(* CFC diagram, written out as Structured Text *)
GVL.s3363[s3363_Mapping.ACV_203].PLC_CMD := RAMP_REAL_1.OUT;
_OR123_OUT := (PVL.Z202_Config.Status.eStatus=eZ202_Status.Recovery_Active_P202) OR (PVL.Z202_Config.Status.eStatus=eZ202_Status.Recovery_Active_P203) OR (PVL.Z202_Config.Status.eStatus=eZ202_Status.Fixed_Rate_Recovery_Active_P202) OR (PVL.Z202_Config.Status.eStatus=eZ202_Status.Fixed_Rate_Recovery_Active_P203) OR (PVL.Z202_Config.Status.eStatus=eZ202_Status.Continuous_Level_And_Recovery_Speed) OR (PVL.Z202_Config.Status.eStatus=eZ202_Status.Continuous_Flow_And_Recovery_Speed) OR (PVL.Z202_Config.Status.eStatus=eZ202_Status.Continuous_Level_And_Recovery_Flow) OR (PVL.Z202_Config.Status.eStatus=eZ202_Status.Continuous_Flow_And_Recovery_Flow);
GVL.s3363[s3363_mapping.ACV_225].PLC_CMD := SEL(PVl.Z202_Config.Valve_Pattern[SubIndex].Matrix.1 AND _OR123_OUT, 0.0, 100);
GVL.s3363[s3363_mapping.ACV_226].PLC_CMD := SEL(_AND161_OUT OR False OR False OR _AND185_OUT, 0.0, 100);
_OR66_OUT := (PVL.Z202_Config.Status.eStatus=eZ202_Status.Opening_ACV203) OR (PVL.Z202_Config.Status.eStatus=eZ202_Status.TK201_Level_Return_Via_P203) OR (PVL.Z202_Config.Status.eStatus=eZ202_Status.Fixed_Rate_Return_Via_P203) OR (PVL.Z202_Config.Status.eStatus=eZ202_Status.Fixed_Rate_Recovery_Active_P203) OR (PVL.Z202_Config.Status.eStatus=eZ202_Status.Recovery_Active_P203) OR (PVL.Z202_Config.Status.eStatus=eZ202_Status.Fixed_Rate_Recovery_Active_P203) OR (PVL.Z202_Config.Status.eStatus=eZ202_Status.Continuous_Level_And_Recovery_Speed) OR (PVL.Z202_Config.Status.eStatus=eZ202_Status.Continuous_Flow_And_Recovery_Speed) OR (PVL.Z202_Config.Status.eStatus=eZ202_Status.Continuous_Level_And_Recovery_Flow) OR (PVL.Z202_Config.Status.eStatus=eZ202_Status.Continuous_Flow_And_Recovery_Flow);
GVL.s3363[s3363_Mapping.ACV_206].PLC_CMD := RAMP_REAL_0.OUT;
RAMP_REAL_0(IN := SEL(_OR241_OUT, 0.0, 100), ASCEND := 50, DESCEND := 5, TIMEBASE := T#1s, RESET := False);
_AND185_OUT := _OR187_OUT AND _OR207_OUT;
_OR187_OUT := (PVL.Z202_Config.Task.eTask=eZ202_Task.TK201_Level_Return_P203) OR (PVL.Z202_Config.Task.eTask=eZ202_Task.Rate_Return_P203) OR (PVL.Z202_Config.Task.eTask=eZ202_Task.Filter_Flow_P203) OR (PVL.Z202_Config.Task.eTask=eZ202_Task.Filter_Level_P203) OR (PVL.Z202_Config.Task.eTask=eZ202_task.Filter_Level_P202_Recovery_Speed_P203) OR (PVL.Z202_Config.Task.eTask=eZ202_task.Filter_Level_P202_Recovery_Flow_P203) OR (PVL.Z202_Config.Task.eTask=eZ202_task.Filter_Flow_P202_Recovery_Speed_P203) OR (PVL.Z202_Config.Task.eTask=eZ202_task.Filter_Flow_P202_Recovery_Flow_P203) OR (PVL.Z202_Config.Task.eTask=eZ202_task.Drain_P203);
_OR48_OUT := (PVL.Z202_Config.Task.eTask=eZ202_Task.TK201_Level_Return_P203) OR (PVL.Z202_Config.Task.eTask=eZ202_Task.Rate_Return_P203) OR (PVL.Z202_Config.Task.eTask=eZ202_Task.Recovery_Rate_P203) OR (PVL.Z202_Config.Task.eTask=eZ202_Task.Recovery_Speed_P203) OR (PVL.Z202_Config.Task.eTask=eZ202_task.Filter_Level_P202_Recovery_Speed_P203) OR (PVL.Z202_Config.Task.eTask=eZ202_task.Filter_Level_P202_Recovery_Flow_P203) OR (PVL.Z202_Config.Task.eTask=eZ202_task.Filter_Flow_P202_Recovery_Speed_P203) OR (PVL.Z202_Config.Task.eTask=eZ202_task.Filter_Flow_P202_Recovery_Flow_P203);
_OR14_OUT := (PVL.Z202_Config.Task.eTask=eZ202_Task.TK201_Level_Return_P202) OR (PVL.Z202_Config.Task.eTask=eZ202_Task.Rate_Return_P202) OR (PVL.Z202_Config.Task.eTask=eZ202_Task.Recovery_Rate_P202) OR (PVL.Z202_Config.Task.eTask=eZ202_Task.Recovery_Speed_P202);
_OR24_OUT := (PVL.Z202_Config.Status.eStatus=eZ202_Status.Opening_ACV203) OR (PVL.Z202_Config.Status.eStatus=eZ202_Status.TK201_Level_Return_Via_P202) OR (PVL.Z202_Config.Status.eStatus=eZ202_Status.Fixed_Rate_Return_Via_P202) OR (PVL.Z202_Config.Status.eStatus=eZ202_Status.Recovery_Active_P202) OR (PVL.Z202_Config.Status.eStatus=eZ202_Status.Fixed_Rate_Recovery_Active_P202);
RAMP_REAL_1(IN := _SEL4_OUT, ASCEND := 50, DESCEND := 5, TIMEBASE := T#1s, RESET := False);
RS_ACV_203();
_SEL4_OUT := SEL((PVL.Z202_Config.Status.eStatus=eZ202_Status.EP101_Level_Return_Via_P203) OR (PVL.Z202_Config.Status.eStatus=eZ202_Status.EP101_Level_Return_Via_P202) OR _OR14_OUT AND _OR24_OUT OR False OR False OR False OR False OR False OR _OR48_OUT AND _OR66_OUT, 0.0, 100);
_OR241_OUT := (PVL.Z202_Config.Status.eStatus=eZ202_Status.EP101_Level_Return_Via_P202) OR False OR False OR False OR False OR _AND253_OUT;
_OR207_OUT := (PVL.Z202_Config.Status.eStatus=eZ202_Status.Opening_ACV206) OR (PVL.Z202_Config.Status.eStatus=eZ202_Status.Opening_ACV203) OR (PVL.Z202_Config.Status.eStatus=eZ202_Status.Opening_ACV226) OR (PVL.Z202_Config.Status.eStatus=eZ202_Status.Fixed_Rate_Return_Via_P203) OR (PVL.Z202_Config.Status.eStatus=eZ202_Status.TK201_Level_Return_Via_P203) OR (PVL.Z202_Config.Status.eStatus=eZ202_Status.Filters_TK201_Level_Control_P203) OR (PVL.Z202_Config.Status.eStatus=eZ202_Status.Filters_Fixed_Flow_Control_P203) OR (PVL.Z202_Config.Status.eStatus=eZ202_Status.Continuous_Level_And_Recovery_Speed) OR (PVL.Z202_Config.Status.eStatus=eZ202_Status.Continuous_Flow_And_Recovery_Speed) OR (PVL.Z202_Config.Status.eStatus=eZ202_Status.Continuous_Level_And_Recovery_Flow) OR (PVL.Z202_Config.Status.eStatus=eZ202_Status.Continuous_Flow_And_Recovery_Flow) OR (PVL.Z202_Config.Status.eStatus=eZ202_Status.Drain_Active_P203);
_AND253_OUT := _OR255_OUT AND _OR271_OUT;
_OR271_OUT := (PVL.Z202_Config.Status.eStatus=eZ202_Status.Opening_ACV206) OR (PVL.Z202_Config.Status.eStatus=eZ202_Status.Opening_ACV203) OR (PVL.Z202_Config.Status.eStatus=eZ202_Status.TK201_Level_Return_Via_P202) OR (PVL.Z202_Config.Status.eStatus=eZ202_Status.Fixed_Rate_Return_Via_P202) OR (PVL.Z202_Config.Status.eStatus=eZ202_Status.Recovery_Active_P202) OR (PVL.Z202_Config.Status.eStatus=eZ202_Status.Fixed_Rate_Recovery_Active_P202) OR (PVL.Z202_Config.Status.eStatus=eZ202_Status.Filters_Fixed_Flow_Control_P203) OR (PVL.Z202_Config.Status.eStatus=eZ202_Status.Filters_TK201_Level_Control_P203) OR (PVL.Z202_Config.Status.eStatus=eZ202_Status.Drain_Active_P203);
_OR255_OUT := (PVL.Z202_Config.Task.eTask=eZ202_Task.TK201_Level_Return_P202) OR (PVL.Z202_Config.Task.eTask=eZ202_Task.Rate_Return_P202) OR (PVL.Z202_Config.Task.eTask=eZ202_Task.Recovery_Rate_P202) OR (PVL.Z202_Config.Task.eTask=eZ202_Task.Recovery_Speed_P202) OR (PVL.Z202_Config.Task.eTask=eZ202_Task.Filter_Flow_P203) OR (PVL.Z202_Config.Task.eTask=eZ202_Task.Filter_Level_P203) OR (PVL.Z202_Config.Task.eTask=eZ202_Task.Drain_P203);
_AND161_OUT := ((PVL.Z202_Config.Task.eTask=eZ202_Task.TK201_Level_Return_P202) OR (PVL.Z202_Config.Task.eTask=eZ202_Task.Rate_Return_P202) OR (PVL.Z202_Config.Task.eTask=eZ202_Task.Filter_Level_P202) OR (PVL.Z202_Config.Task.eTask=eZ202_Task.Filter_Flow_P202) OR (PVL.Z202_Config.Task.eTask=eZ202_Task.Drain_P202)) AND _OR164_OUT;
_OR164_OUT := (PVL.Z202_Config.Status.eStatus=eZ202_Status.Opening_ACV206) OR (PVL.Z202_Config.Status.eStatus=eZ202_Status.Opening_ACV203) OR (PVL.Z202_Config.Status.eStatus=eZ202_Status.Opening_ACV226) OR (PVL.Z202_Config.Status.eStatus=eZ202_Status.TK201_Level_Return_Via_P202) OR (PVL.Z202_Config.Status.eStatus=eZ202_Status.Fixed_Rate_Return_Via_P202) OR (PVL.Z202_Config.Status.eStatus=eZ202_Status.Filters_TK201_Level_Control_P202) OR (PVL.Z202_Config.Status.eStatus=eZ202_Status.Filters_Fixed_Flow_Control_P202) OR (PVL.Z202_Config.Status.eStatus=eZ202_Status.Drain_Active_P202);
GVL.s3363[s3363_mapping.ACV_224].PLC_CMD := SEL(PVl.Z202_Config.Valve_Pattern[SubIndex].Matrix.0 AND ((PVL.Z202_Config.Status.eStatus=eZ202_Status.Recovery_Active_P202) OR (PVL.Z202_Config.Status.eStatus=eZ202_Status.Recovery_Active_P203) OR (PVL.Z202_Config.Status.eStatus=eZ202_Status.Fixed_Rate_Recovery_Active_P202) OR (PVL.Z202_Config.Status.eStatus=eZ202_Status.Fixed_Rate_Recovery_Active_P203) OR (PVL.Z202_Config.Status.eStatus=eZ202_Status.Continuous_Level_And_Recovery_Speed) OR (PVL.Z202_Config.Status.eStatus=eZ202_Status.Continuous_Flow_And_Recovery_Speed) OR (PVL.Z202_Config.Status.eStatus=eZ202_Status.Continuous_Level_And_Recovery_Flow) OR (PVL.Z202_Config.Status.eStatus=eZ202_Status.Continuous_Flow_And_Recovery_Flow)), 0.0, 100);
(* drawn but not wired to any output: PVL.PID[PID_Mapping.Z202_Flow].Actual>5, 50 *)
END_ACTION

ACTION Test_P202_Conflict:
                (*
CASE PVL.Z202_Config.P202_Task.eTask OF
	eZ202_Task.EP101_Level_Return_P202:
		CASE PVl.Z202_Config.P203_Task.eTask OF
			eZ202_Task.EP101_Level_Return_P203:PVL.Z202_Config.P203_Task.eTask:=eZ202_Task.Off;
			eZ202_Task.Filter_Flow_P203:
			eZ202_Task.Filter_Level_P203:
			eZ202_Task.Rate_Return_P203:PVL.Z202_Config.P203_Task.eTask:=eZ202_Task.Off;
			eZ202_Task.Recovery_Rate_P203:PVL.Z202_Config.P203_Task.eTask:=eZ202_Task.Off;
			eZ202_Task.Recovery_Speed_P203:PVL.Z202_Config.P203_Task.eTask:=eZ202_Task.Off;
			eZ202_Task.TK201_Level_Return_P203:PVL.Z202_Config.P203_Task.eTask:=eZ202_Task.Off;
		END_CASE
	eZ202_Task.Filter_Flow_P202:
		CASE PVl.Z202_Config.P203_Task.eTask OF
			eZ202_Task.EP101_Level_Return_P203:
			eZ202_Task.Filter_Flow_P203:PVL.Z202_Config.P203_Task.eTask:=eZ202_Task.Off;
			eZ202_Task.Filter_Level_P203:PVL.Z202_Config.P203_Task.eTask:=eZ202_Task.Off;
			eZ202_Task.Rate_Return_P203:
			eZ202_Task.Recovery_Rate_P203:
			eZ202_Task.Recovery_Speed_P203:
			eZ202_Task.TK201_Level_Return_P203:
		END_CASE
	eZ202_Task.Filter_Level_P202:
		CASE PVl.Z202_Config.P203_Task.eTask OF
			eZ202_Task.EP101_Level_Return_P203:
			eZ202_Task.Filter_Flow_P203:PVL.Z202_Config.P203_Task.eTask:=eZ202_Task.Off;
			eZ202_Task.Filter_Level_P203:PVL.Z202_Config.P203_Task.eTask:=eZ202_Task.Off;
			eZ202_Task.Rate_Return_P203:
			eZ202_Task.Recovery_Rate_P203:
			eZ202_Task.Recovery_Speed_P203:
			eZ202_Task.TK201_Level_Return_P203:
		END_CASE
	eZ202_Task.Rate_Return_P202:
		CASE PVl.Z202_Config.P203_Task.eTask OF
			eZ202_Task.EP101_Level_Return_P203:PVL.Z202_Config.P203_Task.eTask:=eZ202_Task.Off;
			eZ202_Task.Filter_Flow_P203:
			eZ202_Task.Filter_Level_P203:
			eZ202_Task.Rate_Return_P203:PVL.Z202_Config.P203_Task.eTask:=eZ202_Task.Off;
			eZ202_Task.Recovery_Rate_P203:PVL.Z202_Config.P203_Task.eTask:=eZ202_Task.Off;
			eZ202_Task.Recovery_Speed_P203:PVL.Z202_Config.P203_Task.eTask:=eZ202_Task.Off;
			eZ202_Task.TK201_Level_Return_P203:PVL.Z202_Config.P203_Task.eTask:=eZ202_Task.Off;
		END_CASE
	eZ202_Task.Recovery_Rate_P202:
		CASE PVl.Z202_Config.P203_Task.eTask OF
			eZ202_Task.EP101_Level_Return_P203:PVL.Z202_Config.P203_Task.eTask:=eZ202_Task.Off;
			eZ202_Task.Filter_Flow_P203:
			eZ202_Task.Filter_Level_P203:
			eZ202_Task.Rate_Return_P203:PVL.Z202_Config.P203_Task.eTask:=eZ202_Task.Off;
			eZ202_Task.Recovery_Rate_P203:PVL.Z202_Config.P203_Task.eTask:=eZ202_Task.Off;
			eZ202_Task.Recovery_Speed_P203:PVL.Z202_Config.P203_Task.eTask:=eZ202_Task.Off;
			eZ202_Task.TK201_Level_Return_P203:PVL.Z202_Config.P203_Task.eTask:=eZ202_Task.Off;
		END_CASE
	eZ202_Task.Recovery_Speed_P202:
		CASE PVl.Z202_Config.P203_Task.eTask OF
			eZ202_Task.EP101_Level_Return_P203:PVL.Z202_Config.P203_Task.eTask:=eZ202_Task.Off;
			eZ202_Task.Filter_Flow_P203:
			eZ202_Task.Filter_Level_P203:
			eZ202_Task.Rate_Return_P203:PVL.Z202_Config.P203_Task.eTask:=eZ202_Task.Off;
			eZ202_Task.Recovery_Rate_P203:PVL.Z202_Config.P203_Task.eTask:=eZ202_Task.Off;
			eZ202_Task.Recovery_Speed_P203:PVL.Z202_Config.P203_Task.eTask:=eZ202_Task.Off;
			eZ202_Task.TK201_Level_Return_P203:PVL.Z202_Config.P203_Task.eTask:=eZ202_Task.Off;
		END_CASE
	eZ202_Task.TK201_Level_Return_P202:
		CASE PVl.Z202_Config.P203_Task.eTask OF
			eZ202_Task.EP101_Level_Return_P203:PVL.Z202_Config.P203_Task.eTask:=eZ202_Task.Off;
			eZ202_Task.Filter_Flow_P203:
			eZ202_Task.Filter_Level_P203:
			eZ202_Task.Rate_Return_P203:PVL.Z202_Config.P203_Task.eTask:=eZ202_Task.Off;
			eZ202_Task.Recovery_Rate_P203:PVL.Z202_Config.P203_Task.eTask:=eZ202_Task.Off;
			eZ202_Task.Recovery_Speed_P203:PVL.Z202_Config.P203_Task.eTask:=eZ202_Task.Off;
			eZ202_Task.TK201_Level_Return_P203:PVL.Z202_Config.P203_Task.eTask:=eZ202_Task.Off;
		END_CASE
	
END_CASE
*)

              
END_ACTION

ACTION Rate_Return_P202:
                IF PVL.Z202_Config.Task.eTask<> Local_Task THEN
	Local_Task:=PVL.Z202_Config.Task.eTask;
	SubIndex:=0;
	Task_ton.IN:=FALSE;
	local_Status:=eZ202_Status.Opening_Valves;
	PVL.Filter_Config.Mode.eMode:=eFilter_Mode.Off;
	PVL.Z202_Config.ETA:=0;
	Level_Ton.PT:=T#10S;
END_IF;

PVL.PID[PID_Mapping.Z202_Flow].PLC_Target:=PVL.Z202_Config.TK201_Return_Rate.Target;




CASE PVL.Z202_Config.Status.eStatus OF
	eZ202_status.Opening_Valves:
		Local_Status:=eZ202_Status.Opening_ACV226;
	eZ202_status.Opening_ACV226:
		IF GVL.s3363[s3363_mapping.ACV_226].Valve_Actual>75 THEN	Local_Status:=eZ202_Status.Opening_ACV206; END_IF;
	eZ202_Status.Opening_ACV206:
		IF GVL.s3363[s3363_Mapping.ACV_206].Valve_Actual>75 THEN Local_Status:=eZ202_Status.Opening_ACV203;END_IF;
	eZ202_Status.Opening_ACV203:
		IF GVL.s3363[s3363_mapping.ACV_203].Valve_Actual>75 THEN local_Status:=eZ202_Status.Fixed_Rate_Return_Via_P202; END_IF;
		
	eZ202_Status.LT101_High_High_Alarm:		IF Level_ton.Q THEN Local_Status:=eZ202_Status.Waiting_For_Level_OK_LT101; END_IF;
	eZ202_Status.LT201_High_High_Alarm:		IF Level_ton.Q THEN Local_Status:=eZ202_Status.Waiting_For_Level_OK_LT201; END_IF;
	eZ202_Status.LT202_Low_Low_Alarm:		IF Level_ton.Q THEN Local_Status:=eZ202_Status.Waiting_For_Level_OK_LT202; END_IF;
	
	
	eZ202_Status.Waiting_For_Level_OK_LT101:	IF PVL.AIT[ait_Mapping.LT_101_P].Status.eStatus=Burkert.eSensor_Status.OK THEN local_Status:=eZ202_Status.Opening_Valves; END_IF;
	eZ202_Status.Waiting_For_Level_OK_LT201:	IF PVL.AIT[ait_Mapping.LT_201].Status.eStatus=Burkert.eSensor_Status.OK THEN local_Status:=eZ202_Status.Opening_Valves; END_IF;
	eZ202_Status.Waiting_For_Level_OK_LT202:	IF PVL.AIT[ait_Mapping.LT_202].Status.eStatus=Burkert.eSensor_Status.OK THEN local_Status:=eZ202_Status.Opening_Valves; END_IF;

END_CASE;





PVL.Z202_Config.Status.eStatus:= Test_Z201_Return_P202(Local_Status);

Status_hold();



	
		
              
END_ACTION

ACTION Recovery_Rate_P202:
                IF PVL.Z202_Config.Task.eTask<> Local_Task THEN
	Local_Task:=PVL.Z202_Config.Task.eTask;
	SubIndex:=0;
	Task_ton.IN:=FALSE;
	Valve_Ton.IN:=FALSE;
	local_Status:=eZ202_Status.Opening_Valves;
END_IF;



PVL.PID[PID_Mapping.Z202_Flow].PLC_Target:=PVL.Z202_Config.Recovery_Rate.Target;

	
	



Task_ton.PT:=TO_TIME(PVL.Z202_Config.Recovery_Duration_Min);	
Task_ton.IN:=PVL.Z202_Config.Status.eStatus=eZ202_Status.Fixed_Rate_Recovery_Active_P202;
	
//Valve_ton.PT:=TO_TIME(PVL.Z202_Config.Valve_Pattern[SubIndex].Duration);
//IF Valve_ton.Q THEN SubIndex:= ((SubIndex+1) MOD 5); END_IF;;
//Valve_Ton.IN:=NOT(Valve_Ton.Q);

CASE PVL.Z202_Config.Status.eStatus OF
	eZ202_status.Opening_Valves:
		Local_Status:=eZ202_Status.Opening_ACV206;
	eZ202_status.Opening_ACV226:
		IF GVL.s3363[s3363_mapping.ACV_226].Valve_Actual>75 THEN	Local_Status:=eZ202_Status.Opening_ACV206; END_IF;
	eZ202_Status.Opening_ACV206:
		IF GVL.s3363[s3363_Mapping.ACV_206].Valve_Actual>75 THEN Local_Status:=eZ202_Status.Opening_ACV203;END_IF;
	eZ202_Status.Opening_ACV203:
		IF GVL.s3363[s3363_mapping.ACV_203].Valve_Actual>75 THEN local_Status:=eZ202_Status.Fixed_Rate_Recovery_Active_P202; END_IF;
	eZ202_Status.Fixed_Rate_Recovery_Active_P202:
		IF Task_Ton.Q THEN	Local_Status:=eZ202_Status.Recovery_P202_Complete;	END_IF;
	eZ202_Status.LT101_High_High_Alarm:		IF Level_ton.Q THEN Local_Status:=eZ202_Status.Waiting_For_Level_OK_LT101; END_IF;
	eZ202_Status.LT201_High_High_Alarm:		IF Level_ton.Q THEN Local_Status:=eZ202_Status.Waiting_For_Level_OK_LT201; END_IF;
	eZ202_Status.LT202_Low_Low_Alarm:		IF Level_ton.Q THEN Local_Status:=eZ202_Status.Waiting_For_Level_OK_LT202; END_IF;
	eZ202_Status.Waiting_For_Level_OK_LT101:	IF PVL.AIT[ait_Mapping.LT_101_P].Status.eStatus=Burkert.eSensor_Status.OK THEN Local_Task:=eZ202_Task.Off; END_IF;
	eZ202_Status.Waiting_For_Level_OK_LT201:	IF PVL.AIT[ait_Mapping.LT_201].Status.eStatus=Burkert.eSensor_Status.OK THEN Local_Task:=eZ202_Task.Off; END_IF;
	eZ202_Status.Waiting_For_Level_OK_LT202:	IF PVL.AIT[ait_Mapping.LT_202].Status.eStatus=Burkert.eSensor_Status.OK THEN Local_Task:=eZ202_Task.Off; END_IF;
		
END_CASE;



PVL.Z202_Config.Status.eStatus:= Test_All(Local_Status);
Status_hold();
              
END_ACTION

ACTION Status_Hold:
                CASE PVL.Z202_Config.Status.eStatus OF
	eZ202_Status.EP101_High_High_Alarm:		local_Status:=PVL.Z202_Config.Status.eStatus;
	eZ202_Status.P202_Intake_Empty:			local_Status:=PVL.Z202_Config.Status.eStatus;
	eZ202_Status.P203_Intake_Empty:			local_Status:=PVL.Z202_Config.Status.eStatus;
	eZ202_Status.PT202_High_Pressure_Alarm:		local_Status:=PVL.Z202_Config.Status.eStatus;
	eZ202_Status.PT202_Low_Pressure_Alarm:		local_Status:=PVL.Z202_Config.Status.eStatus;
	eZ202_Status.PT203_high_Pressure_Alarm:		local_Status:=PVL.Z202_Config.Status.eStatus;
	eZ202_Status.PT203_Low_Pressure_Alarm:		local_Status:=PVL.Z202_Config.Status.eStatus;
	eZ202_Status.PT202_Not_Ready:				local_Status:=PVL.Z202_Config.Status.eStatus;
	eZ202_Status.PT203_Not_Ready:				local_Status:=PVL.Z202_Config.Status.eStatus;
	eZ202_Status.LT202_Not_Ready:				local_Status:=PVL.Z202_Config.Status.eStatus;
	eZ202_Status.LT202A_Not_Ready:				local_Status:=PVL.Z202_Config.Status.eStatus;
	
	eZ202_Status.FT202_High_High_Flow_Alarm:				local_Status:=PVL.Z202_Config.Status.eStatus;
	ez202_Status.FT202_Low_Low_Flow_Alarm:				local_Status:=PVL.Z202_Config.Status.eStatus;
	eZ202_Status.FT203_High_High_Flow_Alarm:				local_Status:=PVL.Z202_Config.Status.eStatus;
	eZ202_Status.FT203_Low_Low_Flow_Alarm:				local_Status:=PVL.Z202_Config.Status.eStatus;
	//eZ202_Status.PT202_High_Pressure_Alarm:				local_Status:=PVL.Z202_Config.Status.eStatus;
	//eZ202_Status.PT202_Low_Pressure_Alarm:				local_Status:=PVL.Z202_Config.Status.eStatus;
	//eZ202_Status.PT203_High_Pressure_Alarm:				local_Status:=PVL.Z202_Config.Status.eStatus;
	//eZ202_Status.PT203_Low_Pressure_Alarm:					local_Status:=PVL.Z202_Config.Status.eStatus;



END_CASE
              
END_ACTION

ACTION Filter_Flow_P202_Recovery_Speed_P203:
                IF PVL.Z202_Config.Task.eTask<> Local_Task THEN
	Local_Task:=PVL.Z202_Config.Task.eTask;
	local_status:=eZ202_Status.Opening_ACV226;
END_IF;


PVL.PID[PID_Mapping.Z202_TK201_Level].PLC_Target:=PVL.Z202_Config.Filter_Level.Target;
PVL.PID[PID_Mapping.Z202_Filter_Flow ].PLC_Target:=PVL.Z202_Config.Filter_Rate.Target;









CASE PVL.Z202_Config.Status.eStatus OF
	eZ202_Status.Opening_ACV226:
		IF GVL.s3363[s3363_mapping.ACV_226].Valve_Actual>75 THEN	Local_Status:=eZ202_Status.Opening_ACV203;	END_IF;
	eZ202_Status.Opening_ACV203:
		IF GVL.s3363[s3363_Mapping.ACV_203].Valve_Actual>75 THEN	local_Status:=eZ202_Status.Continuous_Flow_And_Recovery_Speed; END_IF;
	eZ202_Status.Continuous_Flow_And_Recovery_Speed:
		IF Task_Ton.Q THEN	PVL.Z202_Config.Task.eTask:=eZ202_Task.Filter_Flow_P202;	END_IF;
	eZ202_Status.LT101_High_High_Alarm:		IF Level_ton.Q THEN Local_Status:=eZ202_Status.Waiting_For_Level_OK_LT101; END_IF;
	eZ202_Status.LT201_High_High_Alarm:		IF Level_ton.Q THEN Local_Status:=eZ202_Status.Waiting_For_Level_OK_LT201; END_IF;
	eZ202_Status.LT202_Low_Low_Alarm:		IF Level_ton.Q THEN Local_Status:=eZ202_Status.Waiting_For_Level_OK_LT202; END_IF;
	eZ202_Status.Waiting_For_Level_OK_LT101:	IF PVL.AIT[ait_Mapping.LT_101_P].Status.eStatus=Burkert.eSensor_Status.OK THEN Local_Task:=eZ202_Task.Off; END_IF;
	eZ202_Status.Waiting_For_Level_OK_LT201:	IF PVL.AIT[ait_Mapping.LT_201].Status.eStatus=Burkert.eSensor_Status.OK THEN Local_Task:=eZ202_Task.Off; END_IF;
	eZ202_Status.Waiting_For_Level_OK_LT202:	IF PVL.AIT[ait_Mapping.LT_202].Status.eStatus=Burkert.eSensor_Status.OK THEN Local_Task:=eZ202_Task.Off; END_IF;

END_CASE




 

//PVL.Z202_Config.Status.eStatus:= Test_Filters(Local_Status);



Task_ton.PT:=TO_TIME(PVL.Z202_Config.Recovery_Duration_Min);	
Task_ton.IN:=PVL.Z202_Config.Status.eStatus=eZ202_Status.Continuous_Flow_And_Recovery_Speed;
	
//Valve_ton.PT:=TO_TIME(PVL.Z202_Config.Valve_Pattern[SubIndex].Duration);
//IF Valve_ton.Q THEN SubIndex:= ((SubIndex+1) MOD 5); END_IF;;
//Valve_Ton.IN:=NOT(Valve_Ton.Q);



PVL.Z202_Config.Status.eStatus:= Test_Combined(local_Status);

Status_hold();
              
END_ACTION

ACTION Filter_Flow_P202_Recovery_Flow_P203:
                IF PVL.Z202_Config.Task.eTask<> Local_Task THEN
	Local_Task:=PVL.Z202_Config.Task.eTask;
	local_status:=eZ202_Status.Opening_ACV226;
END_IF;


PVL.PID[PID_Mapping.Z202_Flow].PLC_Target:=PVL.Z202_Config.Recovery_Rate.Target;
PVL.PID[PID_Mapping.Z202_Filter_Flow ].PLC_Target:=PVL.Z202_Config.Filter_Rate.Target;









CASE PVL.Z202_Config.Status.eStatus OF
	eZ202_Status.Opening_ACV226:
		IF GVL.s3363[s3363_mapping.ACV_226].Valve_Actual>75 THEN	Local_Status:=eZ202_Status.Opening_ACV203;	END_IF;
	eZ202_Status.Opening_ACV203:
		IF GVL.s3363[s3363_Mapping.ACV_203].Valve_Actual>75 THEN	local_Status:=eZ202_Status.Continuous_Flow_And_Recovery_Speed; END_IF;
	eZ202_Status.Continuous_Flow_And_Recovery_Speed:
		IF Task_Ton.Q THEN	PVL.Z202_Config.Task.eTask:=eZ202_Task.Filter_Flow_P202;	END_IF;
		
	eZ202_Status.LT101_High_High_Alarm:		IF Level_ton.Q THEN Local_Status:=eZ202_Status.Waiting_For_Level_OK_LT101; END_IF;
	eZ202_Status.LT201_High_High_Alarm:		IF Level_ton.Q THEN Local_Status:=eZ202_Status.Waiting_For_Level_OK_LT201; END_IF;
	eZ202_Status.LT202_Low_Low_Alarm:		IF Level_ton.Q THEN Local_Status:=eZ202_Status.Waiting_For_Level_OK_LT202; END_IF;
	eZ202_Status.Waiting_For_Level_OK_LT101:	IF PVL.AIT[ait_Mapping.LT_101_P].Status.eStatus=Burkert.eSensor_Status.OK THEN Local_Task:=eZ202_Task.Off; END_IF;
	eZ202_Status.Waiting_For_Level_OK_LT201:	IF PVL.AIT[ait_Mapping.LT_201].Status.eStatus=Burkert.eSensor_Status.OK THEN Local_Task:=eZ202_Task.Off; END_IF;
	eZ202_Status.Waiting_For_Level_OK_LT202:	IF PVL.AIT[ait_Mapping.LT_202].Status.eStatus=Burkert.eSensor_Status.OK THEN Local_Task:=eZ202_Task.Off; END_IF;

END_CASE




 





Task_ton.PT:=TO_TIME(PVL.Z202_Config.Recovery_Duration_Min);	
Task_ton.IN:=PVL.Z202_Config.Status.eStatus=eZ202_Status.Recovery_Active_P203;
	





PVL.Z202_Config.Status.eStatus:= Test_Combined(local_Status);



Status_hold();
              
END_ACTION

ACTION Alarms:
                PVL.Z202_Config.READY:=(Local_Status=PVl.Z202_Config.Status.eStatus);

CASE PVL.Z202_Config.Task.eTask OF
	eZ202_task.Off:
		PVL.AIT[AIT_Mapping.LT_202A].Alarm_Config.Silence:=FALSE;
		PVL.AIT[AIT_MApping.LT_202].Alarm_Config.Silence:=FALSE;
		PVL.s8312[s8312_mapping.PT_202].Alarm_Config.Silence:=TRUE;
		PVL.s8312[s8312_mapping.PT_203].Alarm_Config.Silence:=TRUE;
		PVL.s8050[s8050_mapping.FT_203A].CND.Alarm_Config.Silence:=TRUE;
		PVL.s8050[s8050_mapping.FT_203A].Temp.Alarm_Config.Silence:=TRUE;
		PVL.s8098[s8098_Mapping.FT_202].PDO.Concentration_1.Alarm_Config.Silence:=TRUE;
		PVL.s8098[s8098_Mapping.FT_202].PDO.Concentration_2.Alarm_Config.Silence:=TRUE;
		PVL.s8098[s8098_Mapping.FT_202].PDO.Totaliser_1.Alarm_Config.Silence:=TRUE;
		PVL.s8098[s8098_Mapping.FT_202].PDO.Totaliser_2.Alarm_Config.Silence:=TRUE;
		PVL.s8098[s8098_Mapping.FT_202].PDO.Temp.Alarm_Config.Silence:=TRUE;
		PVL.s8098[s8098_Mapping.FT_202].PDO.VolumeFlow.Alarm_Config.Silence:=TRUE;
		PVL.s8098[s8098_Mapping.FT_203].PDO.Concentration_1.Alarm_Config.Silence:=TRUE;
		PVL.s8098[s8098_Mapping.FT_203].PDO.Concentration_2.Alarm_Config.Silence:=TRUE;
		PVL.s8098[s8098_Mapping.FT_203].PDO.Totaliser_1.Alarm_Config.Silence:=TRUE;
		PVL.s8098[s8098_Mapping.FT_203].PDO.Totaliser_2.Alarm_Config.Silence:=TRUE;
		PVL.s8098[s8098_Mapping.FT_203].PDO.Temp.Alarm_Config.Silence:=TRUE;
		PVL.s8098[s8098_Mapping.FT_203].PDO.VolumeFlow.Alarm_Config.Silence:=TRUE;
	eZ202_Task.Drain_P202:
		PVL.AIT[AIT_Mapping.LT_202A].Alarm_Config.Silence:=FALSE;
		PVL.AIT[AIT_MApping.LT_202].Alarm_Config.Silence:=FALSE;
		PVL.s8312[s8312_mapping.PT_202].Alarm_Config.Silence:=(network.VFD[VFD_Mapping.VFD_202].Output_Pct<Min_Pump_Speed);
		PVL.s8312[s8312_mapping.PT_203].Alarm_Config.Silence:=TRUE;			
		PVL.s8050[s8050_mapping.FT_203A].CND.Alarm_Config.Silence:=TRUE;
		PVL.s8050[s8050_mapping.FT_203A].Temp.Alarm_Config.Silence:=TRUE;
		PVL.s8098[s8098_Mapping.FT_202].PDO.Concentration_1.Alarm_Config.Silence:=TRUE;
		PVL.s8098[s8098_Mapping.FT_202].PDO.Concentration_2.Alarm_Config.Silence:=TRUE;
		PVL.s8098[s8098_Mapping.FT_202].PDO.Totaliser_1.Alarm_Config.Silence:=TRUE;
		PVL.s8098[s8098_Mapping.FT_202].PDO.Totaliser_2.Alarm_Config.Silence:=TRUE;
		PVL.s8098[s8098_Mapping.FT_202].PDO.Temp.Alarm_Config.Silence:=TRUE;
		PVL.s8098[s8098_Mapping.FT_202].PDO.VolumeFlow.Alarm_Config.Silence:=(network.VFD[VFD_Mapping.VFD_202].Output_Pct<Min_Pump_Speed);
		PVL.s8098[s8098_Mapping.FT_203].PDO.Concentration_1.Alarm_Config.Silence:=TRUE;
		PVL.s8098[s8098_Mapping.FT_203].PDO.Concentration_2.Alarm_Config.Silence:=TRUE;
		PVL.s8098[s8098_Mapping.FT_203].PDO.Totaliser_1.Alarm_Config.Silence:=TRUE;
		PVL.s8098[s8098_Mapping.FT_203].PDO.Totaliser_2.Alarm_Config.Silence:=TRUE;
		PVL.s8098[s8098_Mapping.FT_203].PDO.Temp.Alarm_Config.Silence:=TRUE;
		PVL.s8098[s8098_Mapping.FT_203].PDO.VolumeFlow.Alarm_Config.Silence:=TRUE;
	eZ202_Task.Drain_P203:
		PVL.AIT[AIT_Mapping.LT_202A].Alarm_Config.Silence:=FALSE;
		PVL.AIT[AIT_MApping.LT_202].Alarm_Config.Silence:=FALSE;
		PVL.s8312[s8312_mapping.PT_202].Alarm_Config.Silence:=(network.VFD[VFD_Mapping.VFD_203].Output_Pct<Min_Pump_Speed);
		PVL.s8312[s8312_mapping.PT_203].Alarm_Config.Silence:=TRUE;			
		PVL.s8050[s8050_mapping.FT_203A].CND.Alarm_Config.Silence:=TRUE;
		PVL.s8050[s8050_mapping.FT_203A].Temp.Alarm_Config.Silence:=TRUE;
		PVL.s8098[s8098_Mapping.FT_202].PDO.Concentration_1.Alarm_Config.Silence:=TRUE;
		PVL.s8098[s8098_Mapping.FT_202].PDO.Concentration_2.Alarm_Config.Silence:=TRUE;
		PVL.s8098[s8098_Mapping.FT_202].PDO.Totaliser_1.Alarm_Config.Silence:=TRUE;
		PVL.s8098[s8098_Mapping.FT_202].PDO.Totaliser_2.Alarm_Config.Silence:=TRUE;
		PVL.s8098[s8098_Mapping.FT_202].PDO.Temp.Alarm_Config.Silence:=TRUE;
		PVL.s8098[s8098_Mapping.FT_202].PDO.VolumeFlow.Alarm_Config.Silence:=(network.VFD[VFD_Mapping.VFD_203].Output_Pct<Min_Pump_Speed);
		PVL.s8098[s8098_Mapping.FT_203].PDO.Concentration_1.Alarm_Config.Silence:=TRUE;
		PVL.s8098[s8098_Mapping.FT_203].PDO.Concentration_2.Alarm_Config.Silence:=TRUE;
		PVL.s8098[s8098_Mapping.FT_203].PDO.Totaliser_1.Alarm_Config.Silence:=TRUE;
		PVL.s8098[s8098_Mapping.FT_203].PDO.Totaliser_2.Alarm_Config.Silence:=TRUE;
		PVL.s8098[s8098_Mapping.FT_203].PDO.Temp.Alarm_Config.Silence:=TRUE;
		PVL.s8098[s8098_Mapping.FT_203].PDO.VolumeFlow.Alarm_Config.Silence:=TRUE;
	eZ202_Task.EP101_Level_Return_P202:
	eZ202_Task.EP101_Level_Return_P203:
	eZ202_Task.Filter_Flow_P202:
		PVL.AIT[AIT_Mapping.LT_202A].Alarm_Config.Silence:=FALSE;
		PVL.AIT[AIT_MApping.LT_202].Alarm_Config.Silence:=FALSE;
		PVL.s8312[s8312_mapping.PT_202].Alarm_Config.Silence:=(network.VFD[VFD_Mapping.VFD_202].Output_Pct<Min_Pump_Speed);
		PVL.s8312[s8312_mapping.PT_203].Alarm_Config.Silence:=TRUE;
			
		PVL.s8050[s8050_mapping.FT_203A].CND.Alarm_Config.Silence:=TRUE;
		PVL.s8050[s8050_mapping.FT_203A].Temp.Alarm_Config.Silence:=TRUE;
		
		PVL.s8098[s8098_Mapping.FT_202].PDO.Concentration_1.Alarm_Config.Silence:=TRUE;
		PVL.s8098[s8098_Mapping.FT_202].PDO.Concentration_2.Alarm_Config.Silence:=TRUE;
		PVL.s8098[s8098_Mapping.FT_202].PDO.Totaliser_1.Alarm_Config.Silence:=TRUE;
		PVL.s8098[s8098_Mapping.FT_202].PDO.Totaliser_2.Alarm_Config.Silence:=TRUE;
		PVL.s8098[s8098_Mapping.FT_202].PDO.Temp.Alarm_Config.Silence:=TRUE;
		PVL.s8098[s8098_Mapping.FT_202].PDO.VolumeFlow.Alarm_Config.Silence:=(network.VFD[VFD_Mapping.VFD_202].Output_Pct<Min_Pump_Speed);
		
		PVL.s8098[s8098_Mapping.FT_203].PDO.Concentration_1.Alarm_Config.Silence:=TRUE;
		PVL.s8098[s8098_Mapping.FT_203].PDO.Concentration_2.Alarm_Config.Silence:=TRUE;
		PVL.s8098[s8098_Mapping.FT_203].PDO.Totaliser_1.Alarm_Config.Silence:=TRUE;
		PVL.s8098[s8098_Mapping.FT_203].PDO.Totaliser_2.Alarm_Config.Silence:=TRUE;
		PVL.s8098[s8098_Mapping.FT_203].PDO.Temp.Alarm_Config.Silence:=TRUE;
		PVL.s8098[s8098_Mapping.FT_203].PDO.VolumeFlow.Alarm_Config.Silence:=TRUE;
	eZ202_Task.Filter_Flow_P203:
		PVL.AIT[AIT_Mapping.LT_202A].Alarm_Config.Silence:=FALSE;
		PVL.AIT[AIT_MApping.LT_202].Alarm_Config.Silence:=FALSE;
		PVL.s8312[s8312_mapping.PT_202].Alarm_Config.Silence:=(network.VFD[VFD_Mapping.VFD_203].Output_Pct<Min_Pump_Speed);
		PVL.s8312[s8312_mapping.PT_203].Alarm_Config.Silence:=TRUE;
			
		PVL.s8050[s8050_mapping.FT_203A].CND.Alarm_Config.Silence:=TRUE;
		PVL.s8050[s8050_mapping.FT_203A].Temp.Alarm_Config.Silence:=TRUE;
		
		PVL.s8098[s8098_Mapping.FT_202].PDO.Concentration_1.Alarm_Config.Silence:=TRUE;
		PVL.s8098[s8098_Mapping.FT_202].PDO.Concentration_2.Alarm_Config.Silence:=TRUE;
		PVL.s8098[s8098_Mapping.FT_202].PDO.Totaliser_1.Alarm_Config.Silence:=TRUE;
		PVL.s8098[s8098_Mapping.FT_202].PDO.Totaliser_2.Alarm_Config.Silence:=TRUE;
		PVL.s8098[s8098_Mapping.FT_202].PDO.Temp.Alarm_Config.Silence:=TRUE;
		PVL.s8098[s8098_Mapping.FT_202].PDO.VolumeFlow.Alarm_Config.Silence:=(network.VFD[VFD_Mapping.VFD_203].Output_Pct<Min_Pump_Speed);
		
		PVL.s8098[s8098_Mapping.FT_203].PDO.Concentration_1.Alarm_Config.Silence:=TRUE;
		PVL.s8098[s8098_Mapping.FT_203].PDO.Concentration_2.Alarm_Config.Silence:=TRUE;
		PVL.s8098[s8098_Mapping.FT_203].PDO.Totaliser_1.Alarm_Config.Silence:=TRUE;
		PVL.s8098[s8098_Mapping.FT_203].PDO.Totaliser_2.Alarm_Config.Silence:=TRUE;
		PVL.s8098[s8098_Mapping.FT_203].PDO.Temp.Alarm_Config.Silence:=TRUE;
		PVL.s8098[s8098_Mapping.FT_203].PDO.VolumeFlow.Alarm_Config.Silence:=TRUE;
		
	eZ202_Task.Filter_Level_P202:
		PVL.AIT[AIT_Mapping.LT_202A].Alarm_Config.Silence:=FALSE;
		PVL.AIT[AIT_MApping.LT_202].Alarm_Config.Silence:=FALSE;
		PVL.s8312[s8312_mapping.PT_202].Alarm_Config.Silence:=(network.VFD[VFD_Mapping.VFD_202].Output_Pct<Min_Pump_Speed);
		PVL.s8312[s8312_mapping.PT_203].Alarm_Config.Silence:=TRUE;
		PVL.s8050[s8050_mapping.FT_203A].CND.Alarm_Config.Silence:=TRUE;
		PVL.s8050[s8050_mapping.FT_203A].Temp.Alarm_Config.Silence:=TRUE;
		PVL.s8098[s8098_Mapping.FT_202].PDO.Concentration_1.Alarm_Config.Silence:=TRUE;
		PVL.s8098[s8098_Mapping.FT_202].PDO.Concentration_2.Alarm_Config.Silence:=TRUE;
		PVL.s8098[s8098_Mapping.FT_202].PDO.Totaliser_1.Alarm_Config.Silence:=TRUE;
		PVL.s8098[s8098_Mapping.FT_202].PDO.Totaliser_2.Alarm_Config.Silence:=TRUE;
		PVL.s8098[s8098_Mapping.FT_202].PDO.Temp.Alarm_Config.Silence:=TRUE;
		PVL.s8098[s8098_Mapping.FT_202].PDO.VolumeFlow.Alarm_Config.Silence:=TRUE;//(network.VFD[VFD_Mapping.VFD_202].Output_Pct<Min_Pump_Speed);
		PVL.s8098[s8098_Mapping.FT_203].PDO.Concentration_1.Alarm_Config.Silence:=TRUE;
		PVL.s8098[s8098_Mapping.FT_203].PDO.Concentration_2.Alarm_Config.Silence:=TRUE;
		PVL.s8098[s8098_Mapping.FT_203].PDO.Totaliser_1.Alarm_Config.Silence:=TRUE;
		PVL.s8098[s8098_Mapping.FT_203].PDO.Totaliser_2.Alarm_Config.Silence:=TRUE;
		PVL.s8098[s8098_Mapping.FT_203].PDO.Temp.Alarm_Config.Silence:=TRUE;
		PVL.s8098[s8098_Mapping.FT_203].PDO.VolumeFlow.Alarm_Config.Silence:=TRUE;
	eZ202_Task.Filter_Level_P203:
		PVL.AIT[AIT_Mapping.LT_202A].Alarm_Config.Silence:=FALSE;
		PVL.AIT[AIT_MApping.LT_202].Alarm_Config.Silence:=FALSE;
		PVL.s8312[s8312_mapping.PT_202].Alarm_Config.Silence:=(network.VFD[VFD_Mapping.VFD_203].Output_Pct<Min_Pump_Speed);
		PVL.s8312[s8312_mapping.PT_203].Alarm_Config.Silence:=TRUE;
		PVL.s8050[s8050_mapping.FT_203A].CND.Alarm_Config.Silence:=TRUE;
		PVL.s8050[s8050_mapping.FT_203A].Temp.Alarm_Config.Silence:=TRUE;
		PVL.s8098[s8098_Mapping.FT_202].PDO.Concentration_1.Alarm_Config.Silence:=TRUE;
		PVL.s8098[s8098_Mapping.FT_202].PDO.Concentration_2.Alarm_Config.Silence:=TRUE;
		PVL.s8098[s8098_Mapping.FT_202].PDO.Totaliser_1.Alarm_Config.Silence:=TRUE;
		PVL.s8098[s8098_Mapping.FT_202].PDO.Totaliser_2.Alarm_Config.Silence:=TRUE;
		PVL.s8098[s8098_Mapping.FT_202].PDO.Temp.Alarm_Config.Silence:=TRUE;
		PVL.s8098[s8098_Mapping.FT_202].PDO.VolumeFlow.Alarm_Config.Silence:=TRUE;//(network.VFD[VFD_Mapping.VFD_203].Output_Pct<Min_Pump_Speed);
		PVL.s8098[s8098_Mapping.FT_203].PDO.Concentration_1.Alarm_Config.Silence:=TRUE;
		PVL.s8098[s8098_Mapping.FT_203].PDO.Concentration_2.Alarm_Config.Silence:=TRUE;
		PVL.s8098[s8098_Mapping.FT_203].PDO.Totaliser_1.Alarm_Config.Silence:=TRUE;
		PVL.s8098[s8098_Mapping.FT_203].PDO.Totaliser_2.Alarm_Config.Silence:=TRUE;
		PVL.s8098[s8098_Mapping.FT_203].PDO.Temp.Alarm_Config.Silence:=TRUE;
		PVL.s8098[s8098_Mapping.FT_203].PDO.VolumeFlow.Alarm_Config.Silence:=TRUE;
	eZ202_Task.Rate_Return_P202:
		PVL.AIT[AIT_Mapping.LT_202A].Alarm_Config.Silence:=FALSE;
		PVL.AIT[AIT_MApping.LT_202].Alarm_Config.Silence:=FALSE;
		PVL.s8312[s8312_mapping.PT_202].Alarm_Config.Silence:=TRUE;
		PVL.s8312[s8312_mapping.PT_203].Alarm_Config.Silence:=(network.VFD[VFD_Mapping.VFD_202].Output_Pct<Min_Pump_Speed);
			
		PVL.s8050[s8050_mapping.FT_203A].CND.Alarm_Config.Silence:=TRUE;
		PVL.s8050[s8050_mapping.FT_203A].Temp.Alarm_Config.Silence:=TRUE;
		
		PVL.s8098[s8098_Mapping.FT_202].PDO.Concentration_1.Alarm_Config.Silence:=TRUE;
		PVL.s8098[s8098_Mapping.FT_202].PDO.Concentration_2.Alarm_Config.Silence:=TRUE;
		PVL.s8098[s8098_Mapping.FT_202].PDO.Totaliser_1.Alarm_Config.Silence:=TRUE;
		PVL.s8098[s8098_Mapping.FT_202].PDO.Totaliser_2.Alarm_Config.Silence:=TRUE;
		PVL.s8098[s8098_Mapping.FT_202].PDO.Temp.Alarm_Config.Silence:=TRUE;
		PVL.s8098[s8098_Mapping.FT_202].PDO.VolumeFlow.Alarm_Config.Silence:=TRUE;
		
		PVL.s8098[s8098_Mapping.FT_203].PDO.Concentration_1.Alarm_Config.Silence:=TRUE;
		PVL.s8098[s8098_Mapping.FT_203].PDO.Concentration_2.Alarm_Config.Silence:=TRUE;
		PVL.s8098[s8098_Mapping.FT_203].PDO.Totaliser_1.Alarm_Config.Silence:=TRUE;
		PVL.s8098[s8098_Mapping.FT_203].PDO.Totaliser_2.Alarm_Config.Silence:=TRUE;
		PVL.s8098[s8098_Mapping.FT_203].PDO.Temp.Alarm_Config.Silence:=TRUE;
		PVL.s8098[s8098_Mapping.FT_203].PDO.VolumeFlow.Alarm_Config.Silence:=(network.VFD[VFD_Mapping.VFD_202].Output_Pct<Min_Pump_Speed);
		Burkert.Alarm_Window_Convert(window:=PVL.Z202_Config.TK201_Return_Rate,Config:=PVL.s8098[s8098_Mapping.FT_203].PDO.VolumeFlow.Alarm_Config);
		
	eZ202_Task.Rate_Return_P203:
		PVL.AIT[AIT_Mapping.LT_202A].Alarm_Config.Silence:=FALSE;
		PVL.AIT[AIT_MApping.LT_202].Alarm_Config.Silence:=FALSE;
		PVL.s8312[s8312_mapping.PT_202].Alarm_Config.Silence:=TRUE;
		PVL.s8312[s8312_mapping.PT_203].Alarm_Config.Silence:=(network.VFD[VFD_Mapping.VFD_203].Output_Pct<Min_Pump_Speed);		
		PVL.s8050[s8050_mapping.FT_203A].CND.Alarm_Config.Silence:=TRUE;
		//PVL.s8050[s8050_mapping.FT_203A].Rate_1.Alarm_Config.Silence:=FALSE;
		PVL.s8050[s8050_mapping.FT_203A].Temp.Alarm_Config.Silence:=TRUE;
		PVL.s8098[s8098_Mapping.FT_202].PDO.Concentration_1.Alarm_Config.Silence:=TRUE;
		PVL.s8098[s8098_Mapping.FT_202].PDO.Concentration_2.Alarm_Config.Silence:=TRUE;
		PVL.s8098[s8098_Mapping.FT_202].PDO.Totaliser_1.Alarm_Config.Silence:=TRUE;
		PVL.s8098[s8098_Mapping.FT_202].PDO.Totaliser_2.Alarm_Config.Silence:=TRUE;
		PVL.s8098[s8098_Mapping.FT_202].PDO.Temp.Alarm_Config.Silence:=TRUE;
		PVL.s8098[s8098_Mapping.FT_202].PDO.VolumeFlow.Alarm_Config.Silence:=TRUE;
		
		PVL.s8098[s8098_Mapping.FT_203].PDO.Concentration_1.Alarm_Config.Silence:=TRUE;
		PVL.s8098[s8098_Mapping.FT_203].PDO.Concentration_2.Alarm_Config.Silence:=TRUE;
		PVL.s8098[s8098_Mapping.FT_203].PDO.Totaliser_1.Alarm_Config.Silence:=TRUE;
		PVL.s8098[s8098_Mapping.FT_203].PDO.Totaliser_2.Alarm_Config.Silence:=TRUE;
		PVL.s8098[s8098_Mapping.FT_203].PDO.Temp.Alarm_Config.Silence:=TRUE;
		PVL.s8098[s8098_Mapping.FT_203].PDO.VolumeFlow.Alarm_Config.Silence:=(network.VFD[VFD_Mapping.VFD_203].Output_Pct<Min_Pump_Speed);
		Burkert.Alarm_Window_Convert(window:=PVL.Z202_Config.TK201_Return_Rate,Config:=PVL.s8098[s8098_Mapping.FT_203].PDO.VolumeFlow.Alarm_Config);
	eZ202_Task.Recovery_Speed_P202:
		PVL.AIT[AIT_Mapping.LT_202A].Alarm_Config.Silence:=FALSE;
		PVL.AIT[AIT_MApping.LT_202].Alarm_Config.Silence:=FALSE;
		PVL.s8312[s8312_mapping.PT_202].Alarm_Config.Silence:=TRUE;
		PVL.s8312[s8312_mapping.PT_203].Alarm_Config.Silence:=(network.VFD[VFD_Mapping.VFD_202].Output_Pct<Min_Pump_Speed);
			
		PVL.s8050[s8050_mapping.FT_203A].CND.Alarm_Config.Silence:=TRUE;
		//PVL.s8050[s8050_mapping.FT_203A].Rate_1.Alarm_Config.Silence:=FALSE;
		PVL.s8050[s8050_mapping.FT_203A].Temp.Alarm_Config.Silence:=TRUE;
		
		PVL.s8098[s8098_Mapping.FT_202].PDO.Concentration_1.Alarm_Config.Silence:=TRUE;
		PVL.s8098[s8098_Mapping.FT_202].PDO.Concentration_2.Alarm_Config.Silence:=TRUE;
		PVL.s8098[s8098_Mapping.FT_202].PDO.Totaliser_1.Alarm_Config.Silence:=TRUE;
		PVL.s8098[s8098_Mapping.FT_202].PDO.Totaliser_2.Alarm_Config.Silence:=TRUE;
		PVL.s8098[s8098_Mapping.FT_202].PDO.Temp.Alarm_Config.Silence:=TRUE;
		PVL.s8098[s8098_Mapping.FT_202].PDO.VolumeFlow.Alarm_Config.Silence:=TRUE;
		
		PVL.s8098[s8098_Mapping.FT_203].PDO.Concentration_1.Alarm_Config.Silence:=TRUE;
		PVL.s8098[s8098_Mapping.FT_203].PDO.Concentration_2.Alarm_Config.Silence:=TRUE;
		PVL.s8098[s8098_Mapping.FT_203].PDO.Totaliser_1.Alarm_Config.Silence:=TRUE;
		PVL.s8098[s8098_Mapping.FT_203].PDO.Totaliser_2.Alarm_Config.Silence:=TRUE;
		PVL.s8098[s8098_Mapping.FT_203].PDO.Temp.Alarm_Config.Silence:=TRUE;
		PVL.s8098[s8098_Mapping.FT_203].PDO.VolumeFlow.Alarm_Config.Silence:=(network.VFD[VFD_Mapping.VFD_202].Output_Pct<Min_Pump_Speed);
	eZ202_Task.Recovery_Speed_P203:
		PVL.AIT[AIT_Mapping.LT_202A].Alarm_Config.Silence:=FALSE;
		PVL.AIT[AIT_MApping.LT_202].Alarm_Config.Silence:=FALSE;
		PVL.s8312[s8312_mapping.PT_202].Alarm_Config.Silence:=TRUE;
		PVL.s8312[s8312_mapping.PT_203].Alarm_Config.Silence:=(network.VFD[VFD_Mapping.VFD_203].Output_Pct<Min_Pump_Speed);
			
		PVL.s8050[s8050_mapping.FT_203A].CND.Alarm_Config.Silence:=TRUE;
		PVL.s8050[s8050_mapping.FT_203A].Rate_1.Alarm_Config.Silence:=FALSE;
		PVL.s8050[s8050_mapping.FT_203A].Temp.Alarm_Config.Silence:=TRUE;
		
		PVL.s8098[s8098_Mapping.FT_202].PDO.Concentration_1.Alarm_Config.Silence:=TRUE;
		PVL.s8098[s8098_Mapping.FT_202].PDO.Concentration_2.Alarm_Config.Silence:=TRUE;
		PVL.s8098[s8098_Mapping.FT_202].PDO.Totaliser_1.Alarm_Config.Silence:=TRUE;
		PVL.s8098[s8098_Mapping.FT_202].PDO.Totaliser_2.Alarm_Config.Silence:=TRUE;
		PVL.s8098[s8098_Mapping.FT_202].PDO.Temp.Alarm_Config.Silence:=TRUE;
		PVL.s8098[s8098_Mapping.FT_202].PDO.VolumeFlow.Alarm_Config.Silence:=TRUE;
		
		PVL.s8098[s8098_Mapping.FT_203].PDO.Concentration_1.Alarm_Config.Silence:=TRUE;
		PVL.s8098[s8098_Mapping.FT_203].PDO.Concentration_2.Alarm_Config.Silence:=TRUE;
		PVL.s8098[s8098_Mapping.FT_203].PDO.Totaliser_1.Alarm_Config.Silence:=TRUE;
		PVL.s8098[s8098_Mapping.FT_203].PDO.Totaliser_2.Alarm_Config.Silence:=TRUE;
		PVL.s8098[s8098_Mapping.FT_203].PDO.Temp.Alarm_Config.Silence:=TRUE;
		PVL.s8098[s8098_Mapping.FT_203].PDO.VolumeFlow.Alarm_Config.Silence:=(network.VFD[VFD_Mapping.VFD_203].Output_Pct<Min_Pump_Speed);
	eZ202_Task.Recovery_Rate_P202:
		PVL.AIT[AIT_Mapping.LT_202A].Alarm_Config.Silence:=FALSE;
		PVL.AIT[AIT_MApping.LT_202].Alarm_Config.Silence:=FALSE;
		PVL.s8312[s8312_mapping.PT_202].Alarm_Config.Silence:=(network.VFD[VFD_Mapping.VFD_202].Output_Pct<Min_Pump_Speed);
		PVL.s8312[s8312_mapping.PT_203].Alarm_Config.Silence:=(network.VFD[VFD_Mapping.VFD_202].Output_Pct<Min_Pump_Speed);
			
		PVL.s8050[s8050_mapping.FT_203A].CND.Alarm_Config.Silence:=TRUE;
		//PVL.s8050[s8050_mapping.FT_203A].Rate_1.Alarm_Config.Silence:=FALSE;
		PVL.s8050[s8050_mapping.FT_203A].Temp.Alarm_Config.Silence:=TRUE;
		
		PVL.s8098[s8098_Mapping.FT_202].PDO.Concentration_1.Alarm_Config.Silence:=TRUE;
		PVL.s8098[s8098_Mapping.FT_202].PDO.Concentration_2.Alarm_Config.Silence:=TRUE;
		PVL.s8098[s8098_Mapping.FT_202].PDO.Totaliser_1.Alarm_Config.Silence:=TRUE;
		PVL.s8098[s8098_Mapping.FT_202].PDO.Totaliser_2.Alarm_Config.Silence:=TRUE;
		PVL.s8098[s8098_Mapping.FT_202].PDO.Temp.Alarm_Config.Silence:=TRUE;
		PVL.s8098[s8098_Mapping.FT_202].PDO.VolumeFlow.Alarm_Config.Silence:=TRUE;
		
		PVL.s8098[s8098_Mapping.FT_203].PDO.Concentration_1.Alarm_Config.Silence:=TRUE;
		PVL.s8098[s8098_Mapping.FT_203].PDO.Concentration_2.Alarm_Config.Silence:=TRUE;
		PVL.s8098[s8098_Mapping.FT_203].PDO.Totaliser_1.Alarm_Config.Silence:=TRUE;
		PVL.s8098[s8098_Mapping.FT_203].PDO.Totaliser_2.Alarm_Config.Silence:=TRUE;
		PVL.s8098[s8098_Mapping.FT_203].PDO.Temp.Alarm_Config.Silence:=TRUE;
		PVL.s8098[s8098_Mapping.FT_203].PDO.VolumeFlow.Alarm_Config.Silence:=(network.VFD[VFD_Mapping.VFD_202].Output_Pct<Min_Pump_Speed);
	eZ202_Task.Recovery_Rate_P203:
		PVL.AIT[AIT_Mapping.LT_202A].Alarm_Config.Silence:=FALSE;
		PVL.AIT[AIT_MApping.LT_202].Alarm_Config.Silence:=FALSE;
		PVL.s8312[s8312_mapping.PT_202].Alarm_Config.Silence:=TRUE;
		PVL.s8312[s8312_mapping.PT_203].Alarm_Config.Silence:=(network.VFD[VFD_Mapping.VFD_203].Output_Pct<Min_Pump_Speed);
			
		PVL.s8050[s8050_mapping.FT_203A].CND.Alarm_Config.Silence:=TRUE;
		//PVL.s8050[s8050_mapping.FT_203A].Rate_1.Alarm_Config.Silence:=FALSE;
		PVL.s8050[s8050_mapping.FT_203A].Temp.Alarm_Config.Silence:=TRUE;
		
		PVL.s8098[s8098_Mapping.FT_202].PDO.Concentration_1.Alarm_Config.Silence:=TRUE;
		PVL.s8098[s8098_Mapping.FT_202].PDO.Concentration_2.Alarm_Config.Silence:=TRUE;
		PVL.s8098[s8098_Mapping.FT_202].PDO.Totaliser_1.Alarm_Config.Silence:=TRUE;
		PVL.s8098[s8098_Mapping.FT_202].PDO.Totaliser_2.Alarm_Config.Silence:=TRUE;
		PVL.s8098[s8098_Mapping.FT_202].PDO.Temp.Alarm_Config.Silence:=TRUE;
		PVL.s8098[s8098_Mapping.FT_202].PDO.VolumeFlow.Alarm_Config.Silence:=TRUE;
		
		PVL.s8098[s8098_Mapping.FT_203].PDO.Concentration_1.Alarm_Config.Silence:=TRUE;
		PVL.s8098[s8098_Mapping.FT_203].PDO.Concentration_2.Alarm_Config.Silence:=TRUE;
		PVL.s8098[s8098_Mapping.FT_203].PDO.Totaliser_1.Alarm_Config.Silence:=TRUE;
		PVL.s8098[s8098_Mapping.FT_203].PDO.Totaliser_2.Alarm_Config.Silence:=TRUE;
		PVL.s8098[s8098_Mapping.FT_203].PDO.Temp.Alarm_Config.Silence:=TRUE;
		PVL.s8098[s8098_Mapping.FT_203].PDO.VolumeFlow.Alarm_Config.Silence:=(network.VFD[VFD_Mapping.VFD_203].Output_Pct<Min_Pump_Speed);
		
	eZ202_Task.TK201_Level_Return_P202:
		PVL.AIT[AIT_Mapping.LT_202A].Alarm_Config.Silence:=FALSE;
		PVL.AIT[AIT_MApping.LT_202].Alarm_Config.Silence:=FALSE;
		PVL.s8312[s8312_mapping.PT_202].Alarm_Config.Silence:=TRUE;
		PVL.s8312[s8312_mapping.PT_203].Alarm_Config.Silence:=(PVL.PID[PID_Mapping.Z202_TK201_Level].CV<10);	
		PVL.s8050[s8050_mapping.FT_203A].CND.Alarm_Config.Silence:=TRUE;
		PVL.s8050[s8050_mapping.FT_203A].Temp.Alarm_Config.Silence:=TRUE;
		PVL.s8098[s8098_Mapping.FT_202].PDO.Concentration_1.Alarm_Config.Silence:=TRUE;
		PVL.s8098[s8098_Mapping.FT_202].PDO.Concentration_2.Alarm_Config.Silence:=TRUE;
		PVL.s8098[s8098_Mapping.FT_202].PDO.Totaliser_1.Alarm_Config.Silence:=TRUE;
		PVL.s8098[s8098_Mapping.FT_202].PDO.Totaliser_2.Alarm_Config.Silence:=TRUE;
		PVL.s8098[s8098_Mapping.FT_202].PDO.Temp.Alarm_Config.Silence:=TRUE;
		PVL.s8098[s8098_Mapping.FT_202].PDO.VolumeFlow.Alarm_Config.Silence:=TRUE;
		PVL.s8098[s8098_Mapping.FT_203].PDO.Concentration_1.Alarm_Config.Silence:=TRUE;
		PVL.s8098[s8098_Mapping.FT_203].PDO.Concentration_2.Alarm_Config.Silence:=TRUE;
		PVL.s8098[s8098_Mapping.FT_203].PDO.Totaliser_1.Alarm_Config.Silence:=TRUE;
		PVL.s8098[s8098_Mapping.FT_203].PDO.Totaliser_2.Alarm_Config.Silence:=TRUE;
		PVL.s8098[s8098_Mapping.FT_203].PDO.Temp.Alarm_Config.Silence:=TRUE;
		PVL.s8098[s8098_Mapping.FT_203].PDO.VolumeFlow.Alarm_Config.Silence:=TRUE;//(PVL.PID[PID_Mapping.Z202_TK201_Level].CV<10);
		//Burkert.Alarm_Window_Convert(window:=PVL.Z202_Config.Drain,Config:=PVL.s8098[s8098_Mapping.FT_203].PDO.VolumeFlow.Alarm_Config);
		Burkert.Alarm_Window_Convert(window:=PVL.Z202_Config.TK201_Return_Rate,Config:=PVL.s8098[s8098_Mapping.FT_203].PDO.VolumeFlow.Alarm_Config);
	eZ202_Task.TK201_Level_Return_P203:
		PVL.AIT[AIT_Mapping.LT_202A].Alarm_Config.Silence:=FALSE;
		PVL.AIT[AIT_MApping.LT_202].Alarm_Config.Silence:=FALSE;
		PVL.s8312[s8312_mapping.PT_202].Alarm_Config.Silence:=TRUE;
		PVL.s8312[s8312_mapping.PT_203].Alarm_Config.Silence:=(PVL.PID[PID_Mapping.Z202_TK201_Level].CV<10);
		PVL.s8050[s8050_mapping.FT_203A].CND.Alarm_Config.Silence:=TRUE;
		PVL.s8050[s8050_mapping.FT_203A].Temp.Alarm_Config.Silence:=TRUE;
		PVL.s8098[s8098_Mapping.FT_202].PDO.Concentration_1.Alarm_Config.Silence:=TRUE;
		PVL.s8098[s8098_Mapping.FT_202].PDO.Concentration_2.Alarm_Config.Silence:=TRUE;
		PVL.s8098[s8098_Mapping.FT_202].PDO.Totaliser_1.Alarm_Config.Silence:=TRUE;
		PVL.s8098[s8098_Mapping.FT_202].PDO.Totaliser_2.Alarm_Config.Silence:=TRUE;
		PVL.s8098[s8098_Mapping.FT_202].PDO.Temp.Alarm_Config.Silence:=TRUE;
		PVL.s8098[s8098_Mapping.FT_202].PDO.VolumeFlow.Alarm_Config.Silence:=TRUE;
		PVL.s8098[s8098_Mapping.FT_203].PDO.Concentration_1.Alarm_Config.Silence:=TRUE;
		PVL.s8098[s8098_Mapping.FT_203].PDO.Concentration_2.Alarm_Config.Silence:=TRUE;
		PVL.s8098[s8098_Mapping.FT_203].PDO.Totaliser_1.Alarm_Config.Silence:=TRUE;
		PVL.s8098[s8098_Mapping.FT_203].PDO.Totaliser_2.Alarm_Config.Silence:=TRUE;
		PVL.s8098[s8098_Mapping.FT_203].PDO.Temp.Alarm_Config.Silence:=TRUE;
		PVL.s8098[s8098_Mapping.FT_203].PDO.VolumeFlow.Alarm_Config.Silence:=True;//(PVL.PID[PID_Mapping.Z202_TK201_Level].CV<10);
		//Burkert.Alarm_Window_Convert(window:=PVL.Z202_Config.Drain,Config:=PVL.s8098[s8098_Mapping.FT_203].PDO.VolumeFlow.Alarm_Config);
		Burkert.Alarm_Window_Convert(window:=PVL.Z202_Config.TK201_Return_Rate,Config:=PVL.s8098[s8098_Mapping.FT_203].PDO.VolumeFlow.Alarm_Config);

	
END_CASE


(*
//FT-203 return

//IF (PVL.Z202_Config.Task.eTask=eZ202_Task.) THEN
//	Burkert.Alarm_Window_Convert(window:=PVL.Z202_Config.TK201_Return_Rate,Config:=PVL.s8098[s8098_Mapping.FT_203].PDO.VolumeFlow.Alarm_Config);
//ELSE
	Burkert.Alarm_Window_Convert(window:=PVL.Z202_Config.Recovery_Rate,Config:=PVL.s8098[s8098_Mapping.FT_203].PDO.VolumeFlow.Alarm_Config);	
//END_IF;


(*//FT-202
IF (PVL.Z202_Config.Task.eTask=eZ202_TAsk.Drain_P202 OR PVL.Z202_Config.Task.eTask=eZ202_TAsk.Drain_P203 ) THEN
	Burkert.Alarm_Window_Convert(window:=PVL.Z202_Config.Drain	,	Config:=PVL.s8098[s8098_Mapping.FT_202].PDO.VolumeFlow.Alarm_Config	)	;
ELSE	 
	Burkert.Alarm_Window_Convert(window:=PVL.Z202_Config.Filter_Rate	,	Config:=PVL.s8098[s8098_Mapping.FT_202].PDO.VolumeFlow.Alarm_Config	)	;
END_IF;
*)
PVL.s8050[s8050_Mapping.FT_202A].Rate_1.Alarm_Config.Silence:=PVL.s8098[s8098_Mapping.FT_202].PDO.VolumeFlow.Alarm_Config.Silence;

*)
PVL.s8050[s8050_Mapping.FT_203A].Rate_1.Alarm_Config.Silence:=PVL.s8098[s8098_Mapping.FT_203].PDO.VolumeFlow.Alarm_Config.Silence;
PVL.s8050[s8050_Mapping.FT_202A].Rate_1.Alarm_Config.Silence:=PVL.s8098[s8098_Mapping.FT_202].PDO.VolumeFlow.Alarm_Config.Silence;
//LT-202


IF NOT((PVL.Z202_Config.Task.eTask=eZ202_Task.TK201_Level_Return_P202 OR PVL.Z202_Config.Task.eTask=eZ202_Task.TK201_Level_Return_P203)) THEN
	tAlarm.Target:=PVL.AIT[AIT_mapping.LT_202].Analog_Scale.Eu_Max * (PVL.Z202_Config.Filter_Level.Target/100);
	tAlarm.Warn_Window:=PVL.AIT[AIT_mapping.LT_202].Analog_Scale.Eu_Max * (PVL.Z202_Config.Filter_Level.Warn_Window/100);
	tAlarm.Alarm_Window:=PVL.AIT[AIT_mapping.LT_202].Analog_Scale.Eu_Max * (PVL.Z202_Config.Filter_Level.Alarm_Window/100);
	tAlarm.Alarm_Delay:=PVL.Z202_Config.Filter_Level.Alarm_Delay;;
	Burkert.Alarm_Window_Convert(window:=tAlarm	,	Config:=PVL.AIT[AIT_Mapping.LT_202].Alarm_Config);
ELSE
	tAlarm.Target:=PVL.AIT[AIT_mapping.LT_202].Analog_Scale.Eu_Max * (PVL.Z202_Config.TK201_Return_Level.Target/100);
	tAlarm.Warn_Window:=PVL.AIT[AIT_mapping.LT_202].Analog_Scale.Eu_Max * (PVL.Z202_Config.TK201_Return_Level.Warn_Window/100);
	tAlarm.Alarm_Window:=PVL.AIT[AIT_mapping.LT_202].Analog_Scale.Eu_Max * (PVL.Z202_Config.TK201_Return_Level.Alarm_Window/100);
	tAlarm.Alarm_Delay:=PVL.Z202_Config.TK201_Return_Level.Alarm_Delay;;
	Burkert.Alarm_Window_Convert(window:=tAlarm,Config:=PVL.AIT[AIT_Mapping.LT_202].Alarm_Config);
END_IF;

              
END_ACTION

ACTION Filter_Flow_P203:
                IF PVL.Z202_Config.Task.eTask<> Local_Task THEN
	Local_Task:=PVL.Z202_Config.Task.eTask;
	local_status:=eZ202_Status.Opening_ACV226;
	PVL.Z202_Config.ETA:=0;
END_IF;


PVL.PID[PID_Mapping.Z202_Filter_Flow ].PLC_Target:=PVL.Z202_Config.Filter_Rate.Target;




	
	
CASE PVL.Z202_Config.Status.eStatus OF
	eZ202_Status.Opening_ACV226:
		IF GVL.s3363[s3363_mapping.ACV_226].Valve_Actual>75 THEN	local_status:=eZ202_Status.Opening_ACV206;	END_IF;
	eZ202_Status.Opening_ACV206:
		IF GVL.s3363[s3363_mapping.ACV_206].Valve_Actual>75 THEN	local_status:=eZ202_Status.Filters_Fixed_Flow_Control_P203;	END_IF;
	
	eZ202_Status.LT101_High_High_Alarm:		IF Level_ton.Q THEN Local_Status:=eZ202_Status.Waiting_For_Level_OK_LT101; END_IF;
	eZ202_Status.LT201_High_High_Alarm:		IF Level_ton.Q THEN Local_Status:=eZ202_Status.Waiting_For_Level_OK_LT201; END_IF;
	eZ202_Status.LT202_Low_Low_Alarm:		IF Level_ton.Q THEN Local_Status:=eZ202_Status.Waiting_For_Level_OK_LT202; END_IF;
	eZ202_Status.Waiting_For_Level_OK_LT101:	IF PVL.AIT[ait_Mapping.LT_101_P].Status.eStatus=Burkert.eSensor_Status.OK THEN Local_Task:=eZ202_Task.Off; END_IF;
	eZ202_Status.Waiting_For_Level_OK_LT201:	IF PVL.AIT[ait_Mapping.LT_201].Status.eStatus=Burkert.eSensor_Status.OK THEN Local_Task:=eZ202_Task.Off; END_IF;
	eZ202_Status.Waiting_For_Level_OK_LT202:	IF PVL.AIT[ait_Mapping.LT_202].Status.eStatus=Burkert.eSensor_Status.OK THEN Local_Task:=eZ202_Task.Off; END_IF;
END_CASE






PVL.Z202_Config.Status.eStatus:= Test_Filters_P203(Local_Status);
Status_hold();
              
END_ACTION

ACTION PID_ctrl:
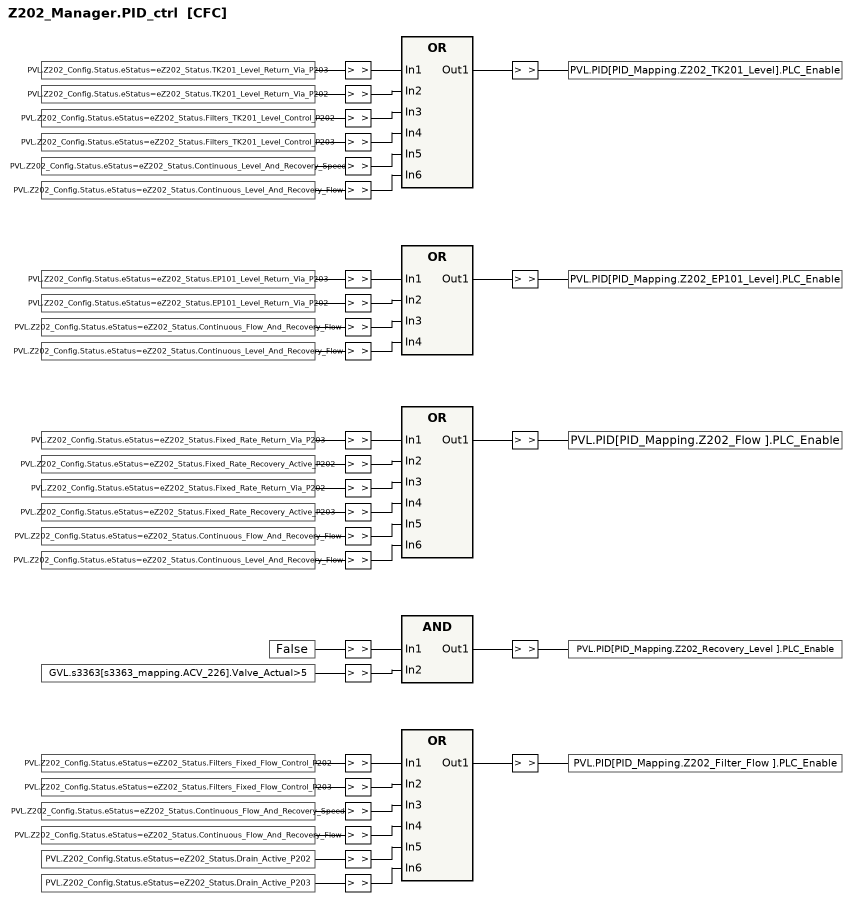
(* [picture p40: Z202_Manager.PID_ctrl, CFC] *)
(* CFC diagram, written out as Structured Text *)
PVL.PID[PID_Mapping.Z202_TK201_Level].PLC_Enable := _OR2_OUT;
PVL.PID[PID_Mapping.Z202_EP101_Level].PLC_Enable := (PVL.Z202_Config.Status.eStatus=eZ202_Status.EP101_Level_Return_Via_P203) OR (PVL.Z202_Config.Status.eStatus=eZ202_Status.EP101_Level_Return_Via_P202) OR (PVL.Z202_Config.Status.eStatus=eZ202_Status.Continuous_Flow_And_Recovery_Flow) OR (PVL.Z202_Config.Status.eStatus=eZ202_Status.Continuous_Level_And_Recovery_Flow);
PVL.PID[PID_Mapping.Z202_Flow ].PLC_Enable := _OR29_OUT;
PVL.PID[PID_Mapping.Z202_Recovery_Level ].PLC_Enable := _AND44_OUT;
PVL.PID[PID_Mapping.Z202_Filter_Flow ].PLC_Enable := (PVL.Z202_Config.Status.eStatus=eZ202_Status.Filters_Fixed_Flow_Control_P202) OR (PVL.Z202_Config.Status.eStatus=eZ202_Status.Filters_Fixed_Flow_Control_P203) OR (PVL.Z202_Config.Status.eStatus=eZ202_Status.Continuous_Flow_And_Recovery_Speed) OR (PVL.Z202_Config.Status.eStatus=eZ202_Status.Continuous_Flow_And_Recovery_Flow) OR (PVL.Z202_Config.Status.eStatus=eZ202_Status.Drain_Active_P202) OR (PVL.Z202_Config.Status.eStatus=eZ202_Status.Drain_Active_P203);
_AND44_OUT := False AND (GVL.s3363[s3363_mapping.ACV_226].Valve_Actual>5);
_OR2_OUT := (PVL.Z202_Config.Status.eStatus=eZ202_Status.TK201_Level_Return_Via_P203) OR (PVL.Z202_Config.Status.eStatus=eZ202_Status.TK201_Level_Return_Via_P202) OR (PVL.Z202_Config.Status.eStatus=eZ202_Status.Filters_TK201_Level_Control_P202) OR (PVL.Z202_Config.Status.eStatus=eZ202_Status.Filters_TK201_Level_Control_P203) OR (PVL.Z202_Config.Status.eStatus=eZ202_Status.Continuous_Level_And_Recovery_Speed) OR (PVL.Z202_Config.Status.eStatus=eZ202_Status.Continuous_Level_And_Recovery_Flow);
_OR29_OUT := (PVL.Z202_Config.Status.eStatus=eZ202_Status.Fixed_Rate_Return_Via_P203) OR (PVL.Z202_Config.Status.eStatus=eZ202_Status.Fixed_Rate_Recovery_Active_P202) OR (PVL.Z202_Config.Status.eStatus=eZ202_Status.Fixed_Rate_Return_Via_P202) OR (PVL.Z202_Config.Status.eStatus=eZ202_Status.Fixed_Rate_Recovery_Active_P203) OR (PVL.Z202_Config.Status.eStatus=eZ202_Status.Continuous_Flow_And_Recovery_Flow) OR (PVL.Z202_Config.Status.eStatus=eZ202_Status.Continuous_Level_And_Recovery_Flow);
END_ACTION

ACTION Rate_Return_P203:
                IF PVL.Z202_Config.Task.eTask<> Local_Task THEN
	Local_Task:=PVL.Z202_Config.Task.eTask;
	SubIndex:=0;
	Task_ton.IN:=FALSE;
	local_Status:=eZ202_Status.Opening_Valves;
	PVL.Z202_Config.ETA:=0;
	PVL.Filter_Config.Mode.eMode:=eFilter_Mode.Off;
END_IF;

PVL.PID[PID_Mapping.Z202_Flow].PLC_Target:=PVL.Z202_Config.TK201_Return_Rate.Target;

	

CASE PVL.Z202_Config.Status.eStatus OF
	eZ202_status.Opening_Valves:
		Local_Status:=eZ202_Status.Opening_ACV226;
	eZ202_Status.Opening_ACV226:
		IF GVL.s3363[s3363_mapping.ACV_226].Valve_Actual>75 THEN Local_Status:=eZ202_Status.Opening_ACV203; END_IF;
	eZ202_Status.Opening_ACV203:
		IF GVL.s3363[s3363_mapping.ACV_203].Valve_Actual>75 THEN local_Status:=eZ202_Status.Fixed_Rate_Return_Via_P203; END_IF;
		
	eZ202_Status.LT101_High_High_Alarm:		IF Level_ton.Q THEN Local_Status:=eZ202_Status.Waiting_For_Level_OK_LT101; END_IF;
	eZ202_Status.LT201_High_High_Alarm:		IF Level_ton.Q THEN Local_Status:=eZ202_Status.Waiting_For_Level_OK_LT201; END_IF;
	eZ202_Status.LT202_Low_Low_Alarm:		IF Level_ton.Q THEN Local_Status:=eZ202_Status.Waiting_For_Level_OK_LT202; END_IF;
	eZ202_Status.Waiting_For_Level_OK_LT101:	IF PVL.AIT[ait_Mapping.LT_101_P].Status.eStatus=Burkert.eSensor_Status.OK THEN Local_Task:=eZ202_Task.Off; END_IF;
	eZ202_Status.Waiting_For_Level_OK_LT201:	IF PVL.AIT[ait_Mapping.LT_201].Status.eStatus=Burkert.eSensor_Status.OK THEN Local_Task:=eZ202_Task.Off; END_IF;
	eZ202_Status.Waiting_For_Level_OK_LT202:	IF PVL.AIT[ait_Mapping.LT_202].Status.eStatus=Burkert.eSensor_Status.OK THEN Local_Task:=eZ202_Task.Off; END_IF;
END_CASE





PVl.Z202_Config.Status.eStatus:= Test_Z201_Return_P203(local_Status);
Status_hold();
              
END_ACTION

ACTION Recovery_Speed_P202:
                Task_ton.IN:=FALSE;
IF PVL.Z202_Config.Task.eTask<> Local_Task THEN
	Local_Task:=PVL.Z202_Config.Task.eTask;
	SubIndex:=0;
	Task_ton.IN:=FALSE;
	Valve_ton.IN:=FALSE;
	Local_Status:=eZ202_Status.Opening_Valves;
	PVL.Filter_Config.Mode.eMode:=eFilter_Mode.Off;
	
END_IF;


	
	


Task_ton.PT:=TO_TIME(PVL.Z202_Config.Recovery_Duration_Min);	
Task_ton.IN:=PVL.Z202_Config.Status.eStatus=eZ202_Status.Recovery_Active_P202;
	
//Valve_ton.PT:=TO_TIME(PVL.Z202_Config.Valve_Pattern[SubIndex].Duration);
//IF Valve_ton.Q THEN SubIndex:= ((SubIndex+1) MOD 5); END_IF;;
//Valve_Ton.IN:=NOT(Valve_Ton.Q);


CASE PVL.Z202_Config.Status.eStatus OF
	eZ202_Status.Opening_Valves:
		Local_Status:=eZ202_Status.Opening_ACV206;
	eZ202_Status.Opening_ACV206:
		IF GVL.s3363[s3363_Mapping.ACV_206].Valve_Actual>75 THEN	local_Status:=eZ202_Status.Opening_ACV203; END_IF;
	eZ202_Status.Opening_ACV203:
		IF GVL.s3363[s3363_Mapping.ACV_203].Valve_Actual>75 THEN	local_Status:=eZ202_Status.Recovery_Active_P202; END_IF;
	eZ202_Status.Recovery_Active_P202:
		IF Task_Ton.Q THEN	Local_Status:=eZ202_Status.Recovery_P202_Complete;	END_IF;
		
	eZ202_Status.LT101_High_High_Alarm:		IF Level_ton.Q THEN Local_Status:=eZ202_Status.Waiting_For_Level_OK_LT101; END_IF;
	eZ202_Status.LT201_High_High_Alarm:		IF Level_ton.Q THEN Local_Status:=eZ202_Status.Waiting_For_Level_OK_LT201; END_IF;
	eZ202_Status.LT202_Low_Low_Alarm:		IF Level_ton.Q THEN Local_Status:=eZ202_Status.Waiting_For_Level_OK_LT202; END_IF;
	eZ202_Status.Waiting_For_Level_OK_LT101:	IF PVL.AIT[ait_Mapping.LT_101_P].Status.eStatus=Burkert.eSensor_Status.OK THEN Local_Task:=eZ202_Task.Off; END_IF;
	eZ202_Status.Waiting_For_Level_OK_LT201:	IF PVL.AIT[ait_Mapping.LT_201].Status.eStatus=Burkert.eSensor_Status.OK THEN Local_Task:=eZ202_Task.Off; END_IF;
	eZ202_Status.Waiting_For_Level_OK_LT202:	IF PVL.AIT[ait_Mapping.LT_202].Status.eStatus=Burkert.eSensor_Status.OK THEN Local_Task:=eZ202_Task.Off; END_IF;
END_CASE;





pvl.Z202_Config.Status.eStatus:= Test_ALL(Local_Status);

Status_hold();
              
END_ACTION

ACTION Filter_Level_P202:
                IF PVL.Z202_Config.Task.eTask<> Local_Task THEN
	Local_Task:=PVL.Z202_Config.Task.eTask;
	local_status:=eZ202_Status.Opening_ACV226;
	PVL.Z202_Config.ETA:=0;
	
END_IF;


PVL.PID[PID_Mapping.Z202_TK201_Level].PLC_Target:=PVL.Z202_Config.Filter_Level.Target;




	
	
CASE PVL.Z202_Config.Status.eStatus OF
	eZ202_Status.Opening_ACV226:
		IF GVL.s3363[s3363_mapping.ACV_226].Valve_Actual>75 THEN	local_status:=eZ202_Status.Filters_TK201_Level_Control_P202;	END_IF;
	eZ202_Status.LT101_High_High_Alarm:		Local_Status:=eZ202_Status.Waiting_For_Level_OK_LT101;
	eZ202_Status.LT201_High_High_Alarm:		Local_Status:=eZ202_Status.Waiting_For_Level_OK_LT201; 
	eZ202_Status.LT202_Low_Low_Alarm:		Local_Status:=eZ202_Status.Waiting_For_Level_OK_LT202;
	eZ202_Status.Waiting_For_Level_OK_LT101:	IF PVL.AIT[ait_Mapping.LT_101_P].Status.eStatus=Burkert.eSensor_Status.OK THEN Local_Task:=eZ202_Task.Off; END_IF;
	eZ202_Status.Waiting_For_Level_OK_LT201:	IF PVL.AIT[ait_Mapping.LT_201].Status.eStatus=Burkert.eSensor_Status.OK THEN Local_Task:=eZ202_Task.Off; END_IF;
	eZ202_Status.Waiting_For_Level_OK_LT202:	IF PVL.AIT[ait_Mapping.LT_202].Status.eStatus=Burkert.eSensor_Status.OK THEN Local_Task:=eZ202_Task.Off; END_IF;
END_CASE




 

PVL.Z202_Config.Status.eStatus:= Test_Filters_P202_LEVEL(Local_Status);

Status_hold();
              
END_ACTION

ACTION Recovery_Speed_P203:
                Task_ton.IN:=FALSE;
IF PVL.Z202_Config.Task.eTask<> Local_Task THEN
	Local_Task:=PVL.Z202_Config.Task.eTask;
	SubIndex:=0;
	Task_ton.IN:=FALSE;
	Valve_ton.IN:=FALSE;
	Local_Status:=eZ202_Status.Opening_Valves;
	PVL.Filter_Config.Mode.eMode:=eFilter_Mode.Off;
	
END_IF;


Task_ton.PT:=TO_TIME(PVL.Z202_Config.Recovery_Duration_Min);	
Task_ton.IN:=PVL.Z202_Config.Status.eStatus=eZ202_Status.Recovery_Active_P203;
	
//Valve_ton.PT:=TO_TIME(PVL.Z202_Config.Valve_Pattern[SubIndex].Duration);
//IF Valve_ton.Q THEN SubIndex:= ((SubIndex+1) MOD 5); END_IF;;
//Valve_Ton.IN:=NOT(Valve_Ton.Q);




CASE PVL.Z202_Config.Status.eStatus OF
	eZ202_Status.Opening_Valves:
		Local_Status:=eZ202_Status.Opening_ACV203;
	eZ202_Status.Opening_ACV203:
		IF GVL.s3363[s3363_Mapping.ACV_203].Valve_Actual>75 THEN	local_Status:=eZ202_Status.Recovery_Active_P203; END_IF;
	eZ202_Status.Recovery_Active_P203:
		IF Task_Ton.Q THEN	Local_Status:=eZ202_Status.Recovery_P203_Complete;	END_IF;
		
	eZ202_Status.LT101_High_High_Alarm:		IF Level_ton.Q THEN Local_Status:=eZ202_Status.Waiting_For_Level_OK_LT101; END_IF;
	eZ202_Status.LT201_High_High_Alarm:		IF Level_ton.Q THEN Local_Status:=eZ202_Status.Waiting_For_Level_OK_LT201; END_IF;
	eZ202_Status.LT202_Low_Low_Alarm:		IF Level_ton.Q THEN Local_Status:=eZ202_Status.Waiting_For_Level_OK_LT202; END_IF;
	eZ202_Status.Waiting_For_Level_OK_LT101:	IF PVL.AIT[ait_Mapping.LT_101_P].Status.eStatus=Burkert.eSensor_Status.OK THEN Local_Task:=eZ202_Task.Off; END_IF;
	eZ202_Status.Waiting_For_Level_OK_LT201:	IF PVL.AIT[ait_Mapping.LT_201].Status.eStatus=Burkert.eSensor_Status.OK THEN Local_Task:=eZ202_Task.Off; END_IF;
	eZ202_Status.Waiting_For_Level_OK_LT202:	IF PVL.AIT[ait_Mapping.LT_202].Status.eStatus=Burkert.eSensor_Status.OK THEN Local_Task:=eZ202_Task.Off; END_IF;
		
END_CASE;





PVL.Z202_Config.Status.eStatus:= Test_ALL(local_Status);
Status_hold();
              
END_ACTION

ACTION Mode_Auto:
                (*
CASE pvl.Z202_Config.P202_Task.eTask OF
	eZ202_Task.Off:
		CASE PVl.Z201_Config.Task.eTask OF
			eZ201_Task.Flow:PVl.Z201_Config.Task.eTask:=eZ201_task.EP101_Level;
		END_CASE;
END_CASE;
CASE pvl.Z202_Config.P203_Task.eTask OF
	eZ202_Task.Off:
		CASE PVl.Z201_Config.Task.eTask OF
			eZ201_Task.Flow:PVl.Z201_Config.Task.eTask:=eZ201_task.EP101_Level;
		END_CASE;
END_CASE;
*)


              
END_ACTION

ACTION TK201_Level_Return_P202:
                IF PVL.Z202_Config.Task.eTask<> Local_Task THEN
	Local_Task:=PVL.Z202_Config.Task.eTask;
	SubIndex:=0;
	Task_ton.IN:=FALSE;
	local_Status:=eZ202_Status.Opening_Valves;
	PVL.Filter_Config.Mode.eMode:=eFilter_Mode.Off;
END_IF;

PVL.PID[PID_Mapping.Z202_TK201_Level].PLC_Target:=PVL.Z202_Config.TK201_Return_Level.Target;




	
	


//Task_ton.PT:=TO_TIME(PVL.Z202_Config.Valve_Pattern[SubIndex].Duration);
//IF Task_ton.Q THEN SubIndex:= ((SubIndex+1) MOD 5); END_IF;;
//Task_ton.IN:=NOT(Task_Ton.Q);

PVL.Z202_Config.ETA:=0;//TO_UDINT(Task_Ton.PT-Task_ton.ET);

CASE PVL.Z202_Config.Status.eStatus OF
	eZ202_status.Opening_Valves:
		Local_Status:=eZ202_Status.Opening_ACV226;
	eZ202_status.Opening_ACV226:
		IF GVL.s3363[s3363_mapping.ACV_226].Valve_Actual>75 THEN	Local_Status:=eZ202_Status.Opening_ACV206; END_IF;
	eZ202_Status.Opening_ACV206:
		IF GVL.s3363[s3363_Mapping.ACV_206].Valve_Actual>75 THEN Local_Status:=eZ202_Status.Opening_ACV203;END_IF;
	eZ202_Status.Opening_ACV203:
		IF GVL.s3363[s3363_mapping.ACV_203].Valve_Actual>75 THEN local_Status:=eZ202_Status.TK201_Level_Return_Via_P202; END_IF;
		
	eZ202_Status.LT101_High_High_Alarm:		IF Level_ton.Q THEN Local_Status:=eZ202_Status.Waiting_For_Level_OK_LT101; END_IF;
	eZ202_Status.LT201_High_High_Alarm:		IF Level_ton.Q THEN Local_Status:=eZ202_Status.Waiting_For_Level_OK_LT201; END_IF;
	eZ202_Status.LT202_Low_Low_Alarm:		IF Level_ton.Q THEN Local_Status:=eZ202_Status.Waiting_For_Level_OK_LT202; END_IF;
	eZ202_Status.Waiting_For_Level_OK_LT101:	IF PVL.AIT[ait_Mapping.LT_101_P].Status.eStatus=Burkert.eSensor_Status.OK THEN Local_Task:=eZ202_Task.Off; END_IF;
	eZ202_Status.Waiting_For_Level_OK_LT201:	IF PVL.AIT[ait_Mapping.LT_201].Status.eStatus=Burkert.eSensor_Status.OK THEN Local_Task:=eZ202_Task.Off; END_IF;
	eZ202_Status.Waiting_For_Level_OK_LT202:	IF PVL.AIT[ait_Mapping.LT_202].Status.eStatus=Burkert.eSensor_Status.OK THEN Local_Task:=eZ202_Task.Off; END_IF;
		
END_CASE;





PVL.Z202_Config.Status.eStatus:= Test_Z201_Return_P202_level(local_Status);

Status_hold();

              
END_ACTION

ACTION Drain_P202:
                IF PVL.Z202_Config.Task.eTask<> Local_Task THEN
	Local_Task:=PVL.Z202_Config.Task.eTask;
	local_status:=eZ202_Status.Opening_ACV226;
	PVL.Z202_Config.ETA:=0;
	PVL.Filter_Config.Mode.eMode:=eFilter_Mode.Off;
END_IF;


PVL.PID[PID_Mapping.Z202_Filter_Flow ].PLC_Target:=PVL.Z202_Config.Drain.Target;

	
	
CASE PVL.Z202_Config.Status.eStatus OF
	eZ202_Status.Opening_ACV226:
		IF GVL.s3363[s3363_mapping.ACV_226].Valve_Actual>90 THEN	local_status:=eZ202_Status.Drain_Active_P202;	END_IF;
	eZ202_Status.P202_Intake_Empty:local_status:=eZ202_Status.Drain_Complete;
	eZ202_Status.Drain_Complete :local_status:=eZ202_Status.Drain_Complete;
	(*
	eZ202_Status.LT101_High_High_Alarm:		IF Level_ton.Q THEN Local_Status:=eZ202_Status.Waiting_For_Level_OK_LT101; END_IF;
	eZ202_Status.LT201_High_High_Alarm:		IF Level_ton.Q THEN Local_Status:=eZ202_Status.Waiting_For_Level_OK_LT201; END_IF;
	eZ202_Status.LT202_Low_Low_Alarm:		IF Level_ton.Q THEN Local_Status:=eZ202_Status.Waiting_For_Level_OK_LT202; END_IF;
	eZ202_Status.Waiting_For_Level_OK_LT101:	IF PVL.AIT[ait_Mapping.LT_101_P].Status.eStatus=Burkert.eSensor_Status.OK THEN Local_Task:=eZ202_Task.Off; END_IF;
	eZ202_Status.Waiting_For_Level_OK_LT201:	IF PVL.AIT[ait_Mapping.LT_201].Status.eStatus=Burkert.eSensor_Status.OK THEN Local_Task:=eZ202_Task.Off; END_IF;
	eZ202_Status.Waiting_For_Level_OK_LT202:	IF PVL.AIT[ait_Mapping.LT_202].Status.eStatus=Burkert.eSensor_Status.OK THEN Local_Task:=eZ202_Task.Off; END_IF;*)
	
END_CASE






PVL.Z202_Config.Status.eStatus:= Test_Drain_P202(Local_Status);
Status_hold();


              
END_ACTION

ACTION Filter_Flow_P202:
                IF PVL.Z202_Config.Task.eTask<> Local_Task THEN
	Local_Task:=PVL.Z202_Config.Task.eTask;
	local_status:=eZ202_Status.Opening_ACV226;
	PVL.Z202_Config.ETA:=0;
END_IF;


PVL.PID[PID_Mapping.Z202_Filter_Flow ].PLC_Target:=PVL.Z202_Config.Filter_Rate.Target;




	
	
CASE PVL.Z202_Config.Status.eStatus OF
	eZ202_Status.Opening_ACV226:
		IF GVL.s3363[s3363_mapping.ACV_226].Valve_Actual>75 THEN	local_status:=eZ202_Status.Filters_Fixed_Flow_Control_P202;	END_IF;
		
	eZ202_Status.LT101_High_High_Alarm:		IF Level_ton.Q THEN Local_Status:=eZ202_Status.Waiting_For_Level_OK_LT101; END_IF;
	eZ202_Status.LT201_High_High_Alarm:		IF Level_ton.Q THEN Local_Status:=eZ202_Status.Waiting_For_Level_OK_LT201; END_IF;
	eZ202_Status.LT202_Low_Low_Alarm:		IF Level_ton.Q THEN Local_Status:=eZ202_Status.Waiting_For_Level_OK_LT202; END_IF;
	eZ202_Status.Waiting_For_Level_OK_LT101:	IF PVL.AIT[ait_Mapping.LT_101_P].Status.eStatus=Burkert.eSensor_Status.OK THEN Local_Task:=eZ202_Task.Off; END_IF;
	eZ202_Status.Waiting_For_Level_OK_LT201:	IF PVL.AIT[ait_Mapping.LT_201].Status.eStatus=Burkert.eSensor_Status.OK THEN Local_Task:=eZ202_Task.Off; END_IF;
	eZ202_Status.Waiting_For_Level_OK_LT202:	IF PVL.AIT[ait_Mapping.LT_202].Status.eStatus=Burkert.eSensor_Status.OK THEN Local_Task:=eZ202_Task.Off; END_IF;
END_CASE






PVL.Z202_Config.Status.eStatus:= Test_Filters_P202(Local_Status);
Status_hold();
              
END_ACTION

ACTION EP101_Level_Return_P203:
                IF PVL.Z202_Config.Task.eTask<> Local_Task THEN
	Local_Task:=PVL.Z202_Config.Task.eTask;
	Task_ton.IN:=FALSE;
	PVL.Filter_Config.Mode.eMode:=eFilter_Mode.Off;
END_IF;

Local_Status:=eZ202_Status.EP101_Level_Return_Via_P203;

PVL.PID[PID_Mapping.Z202_EP101_Level].PLC_Target:=PVL.Z202_Config.EP101_Return_Level.Target;

	


Task_ton.PT:=TO_TIME(PVL.Z202_Config.Valve_Pattern[SubIndex].Duration);
IF Task_ton.Q THEN SubIndex:= ((SubIndex+1) MOD 5); END_IF;;
Task_ton.IN:=NOT(Task_Ton.Q);

PVL.Z202_Config.ETA:=TO_UDINT(Task_Ton.PT-Task_ton.ET);



CASE PVL.Z202_Config.Status.eStatus OF
	eZ202_Status.LT101_High_High_Alarm:		IF Level_ton.Q THEN Local_Status:=eZ202_Status.Waiting_For_Level_OK_LT101; END_IF;
	eZ202_Status.LT201_High_High_Alarm:		IF Level_ton.Q THEN Local_Status:=eZ202_Status.Waiting_For_Level_OK_LT201; END_IF;
	eZ202_Status.LT202_Low_Low_Alarm:		IF Level_ton.Q THEN Local_Status:=eZ202_Status.Waiting_For_Level_OK_LT202; END_IF;
	eZ202_Status.Waiting_For_Level_OK_LT101:	IF PVL.AIT[ait_Mapping.LT_101_P].Status.eStatus=Burkert.eSensor_Status.OK THEN Local_Task:=eZ202_Task.Off; END_IF;
	eZ202_Status.Waiting_For_Level_OK_LT201:	IF PVL.AIT[ait_Mapping.LT_201].Status.eStatus=Burkert.eSensor_Status.OK THEN Local_Task:=eZ202_Task.Off; END_IF;
	eZ202_Status.Waiting_For_Level_OK_LT202:	IF PVL.AIT[ait_Mapping.LT_202].Status.eStatus=Burkert.eSensor_Status.OK THEN Local_Task:=eZ202_Task.Off; END_IF;
END_CASE


PVL.Z202_Config.Status.eStatus:= Test_ALL(Local_Status);
Status_hold();
              
END_ACTION

ACTION Aux:
                Task_Ton();
Valve_Ton();
level_ton();

GVL.Filter_permissive:=(
	PVl.Z202_Config.task.eTask	=	eZ202_Task.Filter_Flow_P202 OR
	PVl.Z202_Config.task.eTask	=	eZ202_Task.Filter_Flow_P202_Recovery_Flow_P203 OR
	PVl.Z202_Config.task.eTask	=	eZ202_Task.Filter_Flow_P202_Recovery_Speed_P203 OR
	PVl.Z202_Config.task.eTask	=	eZ202_Task.Filter_Flow_P203 OR
	PVl.Z202_Config.task.eTask	=	eZ202_Task.Filter_Level_P202 OR
	PVl.Z202_Config.task.eTask	=	eZ202_Task.Filter_Level_P202_Recovery_Flow_P203 OR
	PVl.Z202_Config.task.eTask	=	eZ202_Task.Filter_Level_P202_Recovery_Speed_P203 OR
	PVl.Z202_Config.task.eTask	=	eZ202_Task.Filter_Level_P203 OR
	PVl.Z202_Config.task.eTask	=	eZ202_Task.Drain_P202 OR
	PVl.Z202_Config.task.eTask	=	eZ202_Task.Drain_P203	OR
	PVl.Z202_Config.task.eTask	=	eZ202_Task.Off);



PVL.Z202_Config.TK201_Volume:= (PVl.Z202_Config.Pond_Area_m2  * PVL.AIT[AIT_Mapping.LT_202].EU) / 100;
PVL.Z202_Config.TK201_Catalyst_Level:=PVL.AIT[AIT_Mapping.LT_202A].EU-PVL.AIT[AIT_Mapping.LT_202].EU;

IF Task_Ton.IN THEN
	PVL.Z202_Config.ETA:=TO_UDINT(Task_Ton.PT-Task_ton.ET);
ELSE
	PVL.Z202_Config.ETA:=0;
END_IF

Level_Ton.IN:=(
	PVL.Z202_Config.Status.eStatus=eZ202_Status.LT101_High_High_Alarm OR
	PVL.Z202_Config.Status.eStatus=eZ202_Status.LT201_High_High_Alarm OR
	PVL.Z202_Config.Status.eStatus=eZ202_Status.LT202_Low_Low_Alarm);
	



IF PVL.s8098[s8098_Mapping.FT_101].PDO.VolumeFlow.EU>0 THEN
	PVL.Z201_Config.uvDT:=(0.06 * PVL.AIT[AIT_Mapping.UV_001].EU * PVL.Z202_Config.Pond_Area_m2) /  PVL.s8098[s8098_Mapping.FT_101].PDO.VolumeFlow.EU;
ELSE
	PVL.Z201_Config.uvDT:=0;
END_IF;


Valve_ton.PT:=TO_TIME(PVL.Z202_Config.Valve_Pattern[SubIndex].Duration);
IF Valve_ton.Q THEN SubIndex:= ((SubIndex+1) MOD 5); END_IF;


lcl_Valve_Matrix.0:=(GVL.s3363[s3363_mapping.ACV_224].Valve_Actual>95);
lcl_Valve_Matrix.1:=(GVL.s3363[s3363_mapping.ACV_225].Valve_Actual>95);

Valve_Ton.IN:=(	lcl_Valve_matrix=PVL.Z202_Config.Valve_Pattern[SubIndex].Matrix AND 
	(	local_Status=eZ202_Status.Continuous_Flow_And_Recovery_Speed OR
		local_Status=eZ202_Status.Recovery_Active_P202 OR
		local_Status=eZ202_Status.Recovery_Active_P203 OR
		local_Status=eZ202_Status.Continuous_Flow_And_Recovery_Speed OR
		local_Status=eZ202_Status.Continuous_Flow_And_Recovery_Speed OR
		local_Status=eZ202_Status.Continuous_Level_And_Recovery_Flow OR	
		local_Status=eZ202_Status.Continuous_Level_And_Recovery_Speed OR
		local_Status=eZ202_Status.Fixed_Rate_Recovery_Active_P202 OR
		local_Status=eZ202_Status.Fixed_Rate_Recovery_Active_P203)
);



FT202_Array_Size:=SIZEOF(GVl.FT202_Ave);
IF GVL.CLK_500ms THEN
	IF FT202_Ave_Index<50 AND PVL.s8098[s8098_Mapping.FT_202].PDO.VolumeFlow.EU> 0 THEN	
		GVl.FT202_Ave[FT202_Ave_Index]:=PVL.s8098[s8098_Mapping.FT_202].PDO.VolumeFlow.EU;
		FT202_Ave_Index:=FT202_Ave_Index+1;
	ELSE
		Burkert.MEM.MemMove(pSource:= ADR(GVl.FT202_Ave[1]), pDestination:=ADR(GVl.FT202_Ave[0]) , uiNumberOfBytes:=(SIZEOF(GVl.FT202_Ave)-4) );
		GVl.FT202_Ave[49]:=PVL.s8098[s8098_Mapping.FT_202].PDO.VolumeFlow.EU;
	END_IF;

	IF FT202_Ave_Index>0 THEN
		FT202_Ave:=Burkert.Burkert_OSCAT_BASIC.ARRAY_AVG (	pt:=ADR(GVl.FT202_Ave),	size:=SIZEOF(GVl.FT202_Ave));
		FT202_Hav:=Burkert.Burkert_OSCAT_BASIC.ARRAY_HAV (	pt:=ADR(GVl.FT202_Ave[0]),size:=TO_UINT(FT202_Ave_Index*4));
	END_IF;
	
END_IF;

IF FT202_Ave=0  THEN 	FT202_Ave_Index:=0; END_IF;
PVl.PID[pid_mapping.Z202_Filter_Flow].Actual:=FT202_Ave;



FT203_Array_Size:=SIZEOF(GVl.FT203_Ave);
IF GVL.CLK_500ms THEN
	IF FT203_Ave_Index<50 AND PVL.s8098[s8098_Mapping.FT_203].PDO.VolumeFlow.EU> 0 THEN	
		GVl.FT203_Ave[FT203_Ave_Index]:=PVL.s8098[s8098_Mapping.FT_203].PDO.VolumeFlow.EU;

		FT203_Ave_Index:=FT203_Ave_Index+1;
	ELSE
		Burkert.MEM.MemMove(pSource:= ADR(GVl.FT203_Ave[1]), pDestination:=ADR(GVl.FT203_Ave[0]) , uiNumberOfBytes:=(SIZEOF(GVl.FT203_Ave)-4) );
		GVl.FT203_Ave[49]:=PVL.s8098[s8098_Mapping.FT_203].PDO.VolumeFlow.EU;
	END_IF;

	IF FT203_Ave_Index>0 THEN
		FT203_Ave:=Burkert.Burkert_OSCAT_BASIC.ARRAY_AVG (	pt:=ADR(GVl.FT203_Ave),	size:=SIZEOF(GVl.FT203_Ave));
		FT203_Hav:=Burkert.Burkert_OSCAT_BASIC.ARRAY_HAV (	pt:=ADR(GVl.FT203_Ave[0]),size:=TO_UINT(FT203_Ave_Index*4));
	END_IF;
	
END_IF;

IF FT203_Ave=0  THEN 	FT203_Ave_Index:=0; END_IF;
PVl.PID[pid_mapping.Z202_Flow].Actual:=FT203_AVE;
              
END_ACTION

ACTION Task_Off:
                Task_ton.IN:=FALSE;
Task_Ton.PT:=T#0S;

IF PVL.Z202_Config.Task.eTask<> Local_Task THEN
	PVL.Filter_Config.Mode.eMode:=eFilter_Mode.Off;
	Local_Task:=PVL.Z202_Config.Task.eTask;
END_IF


IF PVL.Z202_Config.Task.eTask=eZ202_Task.Off THEN 
	PVl.Z202_Config.Status.eStatus:= Test_ALL(Local_Status); 
	Local_Task:=PVL.Z202_Config.Task.eTask;
	Local_Status:=eZ202_Status.Off;
	

END_IF;
(*
IF PVL.Z202_Config.P203_Task.eTask=eZ202_Task.Off THEN 
	PVl.Z202_Config.P203_Status.eStatus:= Test_ALL(P203_Local_Status); 
	P203_Local_Task:=PVL.Z202_Config.P203_Task.eTask;
	P203_Local_Status:=eZ202_Status.Off;
END_IF;
*)
              
END_ACTION

ACTION Filter_Level_P202_Recovery_Flow_P203:
                IF PVL.Z202_Config.Task.eTask<> Local_Task THEN
	Local_Task:=PVL.Z202_Config.Task.eTask;
	local_status:=eZ202_Status.Opening_ACV226;
END_IF;


PVL.PID[PID_Mapping.Z202_Flow].PLC_Target:=PVL.Z202_Config.Recovery_Rate.Target;





	
	
CASE PVL.Z202_Config.Status.eStatus OF
	eZ202_Status.Opening_ACV226:
		IF GVL.s3363[s3363_mapping.ACV_226].Valve_Actual>75 THEN	Local_Status:=eZ202_Status.Opening_ACV203;	END_IF;
	eZ202_Status.Opening_ACV203:
		IF GVL.s3363[s3363_Mapping.ACV_203].Valve_Actual>75 THEN	local_Status:=eZ202_Status.Continuous_Level_And_Recovery_Flow; END_IF;
	eZ202_Status.Continuous_Level_And_Recovery_Flow:
		IF Task_Ton.Q THEN	PVL.Z202_Config.Task.eTask:=eZ202_Task.Filter_Level_P202;	END_IF;
	eZ202_Status.LT101_High_High_Alarm:		IF Level_ton.Q THEN Local_Status:=eZ202_Status.Waiting_For_Level_OK_LT101; END_IF;
	eZ202_Status.LT201_High_High_Alarm:		IF Level_ton.Q THEN Local_Status:=eZ202_Status.Waiting_For_Level_OK_LT201; END_IF;
	eZ202_Status.LT202_Low_Low_Alarm:		IF Level_ton.Q THEN Local_Status:=eZ202_Status.Waiting_For_Level_OK_LT202; END_IF;
	eZ202_Status.Waiting_For_Level_OK_LT101:	IF PVL.AIT[ait_Mapping.LT_101_P].Status.eStatus=Burkert.eSensor_Status.OK THEN Local_Task:=eZ202_Task.Off; END_IF;
	eZ202_Status.Waiting_For_Level_OK_LT201:	IF PVL.AIT[ait_Mapping.LT_201].Status.eStatus=Burkert.eSensor_Status.OK THEN Local_Task:=eZ202_Task.Off; END_IF;
	eZ202_Status.Waiting_For_Level_OK_LT202:	IF PVL.AIT[ait_Mapping.LT_202].Status.eStatus=Burkert.eSensor_Status.OK THEN Local_Task:=eZ202_Task.Off; END_IF;

END_CASE




 

//PVL.Z202_Config.Status.eStatus:= Test_Filters(Local_Status);



Task_ton.PT:=TO_TIME(PVL.Z202_Config.Recovery_Duration_Min);	
Task_ton.IN:=PVL.Z202_Config.Status.eStatus=eZ202_Status.Continuous_Level_And_Recovery_Flow;
	
//Valve_ton.PT:=TO_TIME(PVL.Z202_Config.Valve_Pattern[SubIndex].Duration);
//IF Valve_ton.Q THEN SubIndex:= ((SubIndex+1) MOD 5); END_IF;;
//Valve_Ton.IN:=NOT(Valve_Ton.Q);



PVL.Z202_Config.Status.eStatus:= Test_Combined_level(local_Status);

Status_hold();
              
END_ACTION

ACTION VFD_ctrl:
(* CFC diagram, written out as Structured Text *)
Network.VFD[VFD_Mapping.VFD_203].PLC_Run := _GT2_OUT;
Network.VFD[VFD_Mapping.VFD_202].PLC_CMD := _SEL80_OUT;
Network.VFD[VFD_Mapping.VFD_202].PLC_Run := _SEL80_OUT > 5;
_MAX122_OUT := MAX(0.0, PVL.PID[PID_Mapping.Z202_Pressure ].CV, PVL.PID[PID_Mapping.Z202_Recovery_Level ].CV, PVL.PID[PID_Mapping.Z202_Flow ].CV, PVL.PID[PID_Mapping.Z202_Filter_Flow ].CV);
_SEL80_OUT := SEL(PVL.Z202_Config.Status.eStatus=eZ202_Status.Recovery_Active_P202, _SEL84_OUT, PVL.Z202_Config.Recovery_Speed.Target);
_SEL84_OUT := SEL((PVL.Z202_Config.Status.eStatus=eZ202_Status.Continuous_Level_And_Recovery_Flow) OR (PVL.Z202_Config.Status.eStatus=eZ202_Status.Continuous_Level_And_Recovery_Speed) OR (PVL.Z202_Config.Status.eStatus=eZ202_Status.Filters_TK201_Level_Control_P202) OR (PVL.Z202_Config.Status.eStatus=eZ202_Status.TK201_Level_Return_Via_P202), SEL(False OR (PVL.Z202_Config.Status.eStatus=eZ202_Status.Fixed_Rate_Recovery_Active_P202) OR (PVL.Z202_Config.Status.eStatus=eZ202_Status.Recovery_Active_P202) OR False OR (PVL.Z202_Config.Status.eStatus=eZ202_Status.EP101_Level_Return_Via_P202) OR (PVL.Z202_Config.Status.eStatus=eZ202_Status.Fixed_Rate_Return_Via_P202) OR (PVL.Z202_Config.Status.eStatus=eZ202_Status.Filters_Fixed_Flow_Control_P202) OR (PVL.Z202_Config.Status.eStatus=eZ202_Status.Continuous_Flow_And_Recovery_Flow) OR (PVL.Z202_Config.Status.eStatus=eZ202_Status.Continuous_Flow_And_Recovery_Speed) OR (PVL.Z202_Config.Status.eStatus=eZ202_Status.Drain_Active_P202) OR False, 0.0, _MAX122_OUT), PVL.PID[PID_Mapping.Z202_TK201_Level ].CV);
_SEL4_OUT_2 := SEL(_OR6_OUT, _SEL14_OUT, PVL.Z202_Config.Recovery_Speed.Target);
_SEL14_OUT := SEL(_AND16_OUT, _SEL30_OUT, PVL.PID[PID_Mapping.Z202_Filter_Flow ].CV);
_OR6_OUT := (PVL.Z202_Config.Status.eStatus=eZ202_Status.Recovery_Active_P203) OR (PVL.Z202_Config.Status.eStatus=eZ202_Status.Continuous_Level_And_Recovery_Speed) OR (PVL.Z202_Config.Status.eStatus=eZ202_Status.Continuous_Flow_And_Recovery_Speed);
_AND16_OUT := _OR18_OUT AND ((PVL.Z202_Config.Status.eStatus=eZ202_Status.Filters_Fixed_Flow_Control_P203) OR (PVL.Z202_Config.Status.eStatus=eZ202_Status.Drain_Active_P203));
_OR18_OUT := (GVL.s3363[s3363_Mapping.ACV_203].Mode.eMode=Burkert.eACV_Modes.Auto) OR (GVL.s3363[s3363_Mapping.ACV_203].Mode.eMode=Burkert.eACV_Modes.Simulate);
Network.VFD[VFD_Mapping.VFD_203].PLC_CMD := _SEL4_OUT_2;
_OR35_OUT := (PVL.Z202_Config.Status.eStatus=eZ202_Status.TK201_Level_Return_Via_P203) OR (PVL.Z202_Config.Status.eStatus=eZ202_Status.EP101_Level_Return_Via_P203) OR (PVL.Z202_Config.Status.eStatus=eZ202_Status.Fixed_Rate_Return_Via_P203) OR (PVL.Z202_Config.Status.eStatus=eZ202_Status.Recovery_Active_P203) OR (PVL.Z202_Config.Status.eStatus=eZ202_Status.Filters_Fixed_Flow_Control_P203) OR (PVL.Z202_Config.Status.eStatus=eZ202_Status.Filters_TK201_Level_Control_P203) OR (PVL.Z202_Config.Status.eStatus=eZ202_Status.Fixed_Rate_Recovery_Active_P203) OR (PVL.Z202_Config.Status.eStatus=eZ202_Status.Continuous_Level_And_Recovery_Flow) OR (PVL.Z202_Config.Status.eStatus=eZ202_Status.Continuous_Flow_And_Recovery_Flow) OR False;
_SEL30_OUT := SEL(_OR18_OUT AND _OR35_OUT, 0.0, MAX(PVL.PID[PID_Mapping.Z202_EP101_Level].CV, PVL.PID[PID_Mapping.Z202_Flow ].CV, PVL.PID[PID_Mapping.Z202_Pressure ].CV, PVL.PID[PID_Mapping.Z202_TK201_Level ].CV, PVL.PID[PID_Mapping.Z202_Recovery_Level ].CV));
_GT2_OUT := _SEL4_OUT_2 > 5;
END_ACTION

ACTION Filter_Level_P202_Recovery_Speed_P203:
                IF PVL.Z202_Config.Task.eTask<> Local_Task THEN
	Local_Task:=PVL.Z202_Config.Task.eTask;
	local_status:=eZ202_Status.Opening_ACV226;
END_IF;


PVL.PID[PID_Mapping.Z202_TK201_Level].PLC_Target:=PVL.Z202_Config.Filter_Level.Target;




	
	
CASE PVL.Z202_Config.Status.eStatus OF
	eZ202_Status.Opening_ACV226:
		IF GVL.s3363[s3363_mapping.ACV_226].Valve_Actual>75 THEN	Local_Status:=eZ202_Status.Opening_ACV203;	END_IF;
	eZ202_Status.Opening_ACV203:
		IF GVL.s3363[s3363_Mapping.ACV_203].Valve_Actual>75 THEN	local_Status:=eZ202_Status.Continuous_Level_And_Recovery_Speed; END_IF;
	eZ202_Status.Continuous_Level_And_Recovery_Speed:
		IF Task_Ton.Q THEN	PVL.Z202_Config.Task.eTask:=eZ202_Task.Filter_Level_P202;	END_IF;
	eZ202_Status.LT101_High_High_Alarm:		IF Level_ton.Q THEN Local_Status:=eZ202_Status.Waiting_For_Level_OK_LT101; END_IF;
	eZ202_Status.LT201_High_High_Alarm:		IF Level_ton.Q THEN Local_Status:=eZ202_Status.Waiting_For_Level_OK_LT201; END_IF;
	eZ202_Status.LT202_Low_Low_Alarm:		IF Level_ton.Q THEN Local_Status:=eZ202_Status.Waiting_For_Level_OK_LT202; END_IF;
	eZ202_Status.Waiting_For_Level_OK_LT101:	IF PVL.AIT[ait_Mapping.LT_101_P].Status.eStatus=Burkert.eSensor_Status.OK THEN Local_Task:=eZ202_Task.Off; END_IF;
	eZ202_Status.Waiting_For_Level_OK_LT201:	IF PVL.AIT[ait_Mapping.LT_201].Status.eStatus=Burkert.eSensor_Status.OK THEN Local_Task:=eZ202_Task.Off; END_IF;
	eZ202_Status.Waiting_For_Level_OK_LT202:	IF PVL.AIT[ait_Mapping.LT_202].Status.eStatus=Burkert.eSensor_Status.OK THEN Local_Task:=eZ202_Task.Off; END_IF;

END_CASE




 

//PVL.Z202_Config.Status.eStatus:= Test_Filters(Local_Status);



Task_ton.PT:=TO_TIME(PVL.Z202_Config.Recovery_Duration_Min);	
Task_ton.IN:=PVL.Z202_Config.Status.eStatus=eZ202_Status.Continuous_Level_And_Recovery_Speed;
	
//Valve_ton.PT:=TO_TIME(PVL.Z202_Config.Valve_Pattern[SubIndex].Duration);//
//IF Valve_ton.Q THEN SubIndex:= ((SubIndex+1) MOD 5); END_IF;;
///Valve_Ton.IN:=NOT(Valve_Ton.Q);


PVL.Z202_Config.Status.eStatus:= Test_Combined_level(local_Status);

Status_hold();
              
END_ACTION

ACTION Drain_P203:
                IF PVL.Z202_Config.Task.eTask<> Local_Task THEN
	Local_Task:=PVL.Z202_Config.Task.eTask;
	local_status:=eZ202_Status.Opening_ACV226;
	PVL.Z202_Config.ETA:=0;
	PVL.Filter_Config.Mode.eMode:=eFilter_Mode.Off;
END_IF;


PVL.PID[PID_Mapping.Z202_Filter_Flow ].PLC_Target:=PVL.Z202_Config.Filter_Rate.Target;




	
	
CASE PVL.Z202_Config.Status.eStatus OF
	eZ202_Status.Opening_ACV226:
		IF GVL.s3363[s3363_mapping.ACV_226].Valve_Actual>75 THEN	local_status:=eZ202_Status.Opening_ACV206;	END_IF;
	eZ202_Status.Opening_ACV206:
		IF GVL.s3363[s3363_mapping.ACV_206].Valve_Actual>75 THEN	local_status:=eZ202_Status.Drain_Active_P203;	END_IF;
	eZ202_Status.P203_Intake_Empty:local_status:=eZ202_Status.Drain_Complete;
	eZ202_Status.Drain_Complete :local_status:=eZ202_Status.Drain_Complete;
END_CASE






PVL.Z202_Config.Status.eStatus:= Test_Drain_P203(Local_Status);
Status_hold();
              
END_ACTION

ACTION Recovery_Rate_P203:
                Task_ton.IN:=FALSE;
IF PVL.Z202_Config.Task.eTask<> Local_Task THEN
	Local_Task:=PVL.Z202_Config.Task.eTask;
	SubIndex:=0;
	Task_ton.IN:=FALSE;
	Valve_ton.IN:=FALSE;
	Local_Status:=eZ202_Status.Opening_Valves;
	PVL.Filter_Config.Mode.eMode:=eFilter_Mode.Off;
	
END_IF;


	
PVL.PID[PID_Mapping.Z202_Flow].PLC_Target:=PVL.Z202_Config.Recovery_Rate.Target;

	
	


Task_ton.PT:=TO_TIME(PVL.Z202_Config.Recovery_Duration_Min);	
Task_ton.IN:=PVL.Z202_Config.Status.eStatus=eZ202_Status.Fixed_Rate_Recovery_Active_P203;
	
//Valve_ton.PT:=TO_TIME(PVL.Z202_Config.Valve_Pattern[SubIndex].Duration);
//IF Valve_ton.Q THEN SubIndex:= ((SubIndex+1) MOD 5); END_IF;;
//Valve_Ton.IN:=NOT(Valve_Ton.Q);


CASE PVL.Z202_Config.Status.eStatus OF
	eZ202_Status.Opening_Valves:
		Local_Status:=eZ202_Status.Opening_ACV203;
	eZ202_Status.Opening_ACV203:
		IF GVL.s3363[s3363_Mapping.ACV_203].Valve_Actual>75 THEN	local_Status:=eZ202_Status.Fixed_Rate_Recovery_Active_P203; END_IF;
	eZ202_Status.Fixed_Rate_Recovery_Active_P203:
		IF Task_Ton.Q THEN	Local_Status:=eZ202_Status.Recovery_P203_Complete;	END_IF;
		
	eZ202_Status.LT101_High_High_Alarm:		IF Level_ton.Q THEN Local_Status:=eZ202_Status.Waiting_For_Level_OK_LT101; END_IF;
	eZ202_Status.LT201_High_High_Alarm:		IF Level_ton.Q THEN Local_Status:=eZ202_Status.Waiting_For_Level_OK_LT201; END_IF;
	eZ202_Status.LT202_Low_Low_Alarm:		IF Level_ton.Q THEN Local_Status:=eZ202_Status.Waiting_For_Level_OK_LT202; END_IF;
	eZ202_Status.Waiting_For_Level_OK_LT101:	IF PVL.AIT[ait_Mapping.LT_101_P].Status.eStatus=Burkert.eSensor_Status.OK THEN Local_Task:=eZ202_Task.Off; END_IF;
	eZ202_Status.Waiting_For_Level_OK_LT201:	IF PVL.AIT[ait_Mapping.LT_201].Status.eStatus=Burkert.eSensor_Status.OK THEN Local_Task:=eZ202_Task.Off; END_IF;
	eZ202_Status.Waiting_For_Level_OK_LT202:	IF PVL.AIT[ait_Mapping.LT_202].Status.eStatus=Burkert.eSensor_Status.OK THEN Local_Task:=eZ202_Task.Off; END_IF;
	
END_CASE;





PVL.Z202_Config.Status.eStatus:= Test_ALL(local_Status);
Status_hold();
              
END_ACTION

ACTION TK201_Level_Return_P203:
                IF PVL.Z202_Config.Task.eTask<> Local_Task THEN
	Local_Task:=PVL.Z202_Config.Task.eTask;
	SubIndex:=0;
	Task_ton.IN:=FALSE;
	local_Status:=eZ202_Status.Opening_Valves;
	PVL.Filter_Config.Mode.eMode:=eFilter_Mode.Off;
END_IF;


PVL.PID[PID_Mapping.Z202_TK201_Level].PLC_Target:=PVL.Z202_Config.TK201_Return_Level.Target;

//Task_ton.PT:=TO_TIME(PVL.Z202_Config.Valve_Pattern[SubIndex].Duration);
//IF Task_ton.Q THEN SubIndex:= ((SubIndex+1) MOD 5); END_IF;;
Task_ton.IN:=FALSE;

PVL.Z202_Config.ETA:=0;


CASE PVL.Z202_Config.Status.eStatus OF
	eZ202_status.Opening_Valves:
		Local_Status:=eZ202_Status.Opening_ACV226;
	eZ202_Status.Opening_ACV226:
		IF GVL.s3363[s3363_mapping.ACV_226].Valve_Actual>75 THEN Local_Status:=eZ202_Status.Opening_ACV203; END_IF;
	eZ202_Status.Opening_ACV203:
		IF GVL.s3363[s3363_mapping.ACV_203].Valve_Actual>75 THEN local_Status:=eZ202_Status.TK201_Level_Return_Via_P203; END_IF;
	eZ202_Status.LT101_High_High_Alarm:		IF Level_ton.Q THEN Local_Status:=eZ202_Status.Waiting_For_Level_OK_LT101; END_IF;
	eZ202_Status.LT201_High_High_Alarm:		IF Level_ton.Q THEN Local_Status:=eZ202_Status.Waiting_For_Level_OK_LT201; END_IF;
	eZ202_Status.LT202_Low_Low_Alarm:		IF Level_ton.Q THEN Local_Status:=eZ202_Status.Waiting_For_Level_OK_LT202; END_IF;
	eZ202_Status.Waiting_For_Level_OK_LT101:	IF PVL.AIT[ait_Mapping.LT_101_P].Status.eStatus=Burkert.eSensor_Status.OK THEN Local_Task:=eZ202_Task.Off; END_IF;
	eZ202_Status.Waiting_For_Level_OK_LT201:	IF PVL.AIT[ait_Mapping.LT_201].Status.eStatus=Burkert.eSensor_Status.OK THEN Local_Task:=eZ202_Task.Off; END_IF;
	eZ202_Status.Waiting_For_Level_OK_LT202:	IF PVL.AIT[ait_Mapping.LT_202].Status.eStatus=Burkert.eSensor_Status.OK THEN Local_Task:=eZ202_Task.Off; END_IF;
		
END_CASE




PVL.Z202_Config.Status.eStatus:= Test_Z201_Return_P203_level(local_Status);
Status_hold();
              
END_ACTION

ACTION Filter_Level_P203:
                IF PVL.Z202_Config.Task.eTask<> Local_Task THEN
	Local_Task:=PVL.Z202_Config.Task.eTask;
	local_status:=eZ202_Status.Opening_ACV226;
	PVL.Z202_Config.ETA:=0;
END_IF;


PVL.PID[PID_Mapping.Z202_TK201_Level].PLC_Target:=PVL.Z202_Config.Filter_Level.Target;




	
	
CASE PVL.Z202_Config.Status.eStatus OF
	eZ202_Status.Opening_ACV226:
		IF GVL.s3363[s3363_mapping.ACV_226].Valve_Actual>75 THEN	local_status:=eZ202_Status.Opening_ACV206;	END_IF;
	eZ202_Status.Opening_ACV206:
		IF GVL.s3363[s3363_mapping.ACV_206].Valve_Actual>75 THEN	local_status:=eZ202_Status.Filters_TK201_Level_Control_P203;	END_IF;
		
	eZ202_Status.LT101_High_High_Alarm:		IF Level_ton.Q THEN Local_Status:=eZ202_Status.Waiting_For_Level_OK_LT101; END_IF;
	eZ202_Status.LT201_High_High_Alarm:		IF Level_ton.Q THEN Local_Status:=eZ202_Status.Waiting_For_Level_OK_LT201; END_IF;
	eZ202_Status.LT202_Low_Low_Alarm:		IF Level_ton.Q THEN Local_Status:=eZ202_Status.Waiting_For_Level_OK_LT202; END_IF;
	eZ202_Status.Waiting_For_Level_OK_LT101:	IF PVL.AIT[ait_Mapping.LT_101_P].Status.eStatus=Burkert.eSensor_Status.OK THEN Local_Task:=eZ202_Task.Off; END_IF;
	eZ202_Status.Waiting_For_Level_OK_LT201:	IF PVL.AIT[ait_Mapping.LT_201].Status.eStatus=Burkert.eSensor_Status.OK THEN Local_Task:=eZ202_Task.Off; END_IF;
	eZ202_Status.Waiting_For_Level_OK_LT202:	IF PVL.AIT[ait_Mapping.LT_202].Status.eStatus=Burkert.eSensor_Status.OK THEN Local_Task:=eZ202_Task.Off; END_IF;
END_CASE




 

PVL.Z202_Config.Status.eStatus:= Test_Filters_P203_level(Local_Status);
Status_hold();
              
END_ACTION

METHOD Test_Filters_P202 : eZ202_Status
  VAR_INPUT
    Status : eZ202_status;
  END_VAR
  VAR
    tStatus : eZ202_Status;
  END_VAR
                  tStatus:=Status;
IF NOT(GVL.Filter_Path_Available) THEN tStatus:=eZ202_Status.No_Filter_Available; END_IF;


//IF NOT(GVL.s3363[s3363_mapping.ACV_203].Ready) 	THEN 	tStatus:=eZ202_Status.ACV203_Not_Ready; 	END_IF;
//IF NOT(GVL.s3363[s3363_mapping.ACV_206].Ready) 	THEN 	tStatus:=eZ202_Status.ACV206_Not_Ready; 	END_IF;
//IF NOT(GVL.s3363[s3363_mapping.ACV_224].Ready) 	THEN 	tStatus:=eZ202_Status.ACV224_Not_Ready; 	END_IF;
//IF NOT(GVL.s3363[s3363_mapping.ACV_225].Ready) 	THEN 	tStatus:=eZ202_Status.ACV225_Not_Ready; 	END_IF;
IF NOT(GVL.s3363[s3363_mapping.ACV_226].Ready) 	THEN 	tStatus:=eZ202_Status.ACV226_Not_Ready; 	END_IF;

IF NOT(Network.VFD[VFD_Mapping.VFD_202].Ready) 	THEN	tStatus:=eZ202_status.P202_Not_Ready;		END_IF;
//IF NOT(Network.VFD[VFD_Mapping.VFD_203].Ready) 	THEN	tStatus:=eZ202_status.P203_Not_Ready;		END_IF;

IF NOT(PVL.Ait[AIT_Mapping.LT_202].Ready) 		THEN	tStatus:=eZ202_Status.LT202_Not_Ready;		END_IF;
//IF NOT(PVL.Ait[AIT_Mapping.LT_202A].Ready) 		THEN	tStatus:=eZ202_Status.LT202A_Not_Ready;		END_IF;

IF NOT(PVl.s8312[s8312_mapping.PT_202].Ready)	THEN	tStatus:=ez202_Status.PT202_Not_Ready;		END_IF;
//IF NOT(PVl.s8312[s8312_mapping.PT_203].Ready)	THEN	tStatus:=ez202_Status.PT203_Not_Ready;		END_IF;

IF NOT(PVL.s8098[s8098_mapping.FT_202].Ready)	THEN	tStatus:=ez202_Status.FT202_Not_Ready;		END_IF;
//IF NOT(PVL.s8098[s8098_mapping.FT_203].Ready)	THEN	tStatus:=ez202_Status.FT203_Not_Ready;		END_IF;
	
IF gvl.LS[ls_mapping.LSLL_205].Status.eStatus=Burkert.DI_Status.No_Liquid_Detected_Alarm	THEN	tStatus:=eZ202_Status.P202_Intake_Empty;		END_IF;
//IF gvl.LS[ls_mapping.LSLL_203].Status.eStatus=Burkert.DI_Status.No_Liquid_Detected_Alarm	THEN	tStatus:=eZ202_Status.P203_Intake_Empty;		END_IF;
//IF gvl.LS[ls_mapping.LSHH_201].Status.eStatus=Burkert.DI_Status.Liquid_Detected_Alarm		THEN	tStatus:=eZ202_Status.EP101_High_High_Alarm;	END_IF;




//IF GVL.s3363[s3363_mapping.ACV_203].Status.eStatus=Burkert.eACV_Status.Pos_Error THEN	tStatus:=eZ202_Status.ACV203_Error; END_IF;
//IF GVL.s3363[s3363_mapping.ACV_206].Status.eStatus=Burkert.eACV_Status.Pos_Error THEN	tStatus:=eZ202_Status.ACV206_Error; END_IF;
//IF GVL.s3363[s3363_mapping.ACV_224].Status.eStatus=Burkert.eACV_Status.Pos_Error THEN	tStatus:=eZ202_Status.ACV224_Error; END_IF;
//IF GVL.s3363[s3363_mapping.ACV_225].Status.eStatus=Burkert.eACV_Status.Pos_Error THEN	tStatus:=eZ202_Status.ACV225_Error; END_IF;
IF GVL.s3363[s3363_mapping.ACV_226].Status.eStatus=Burkert.eACV_Status.Pos_Error THEN	tStatus:=eZ202_Status.ACV226_Error; END_IF;


IF PVL.AIT[AIT_Mapping.LT_202].Status.eStatus=Burkert.eSensor_Status.Low_Low_Alarm THEN	tStatus:=eZ202_Status.LT202_Low_Low_Alarm;	END_IF;
//IF PVL.AIT[AIT_Mapping.LT_202A].Status.eStatus=Burkert.eSensor_Status.Low_Low_Alarm THEN	tStatus:=eZ202_Status.LT202A_Low_Low_Alarm;	END_IF;

IF (PVL.s8098[s8098_mapping.FT_202].PDO.VolumeFlow.Status.eStatus=burkert.eSensor_Status.Low_Low_Alarm)	THEN	tStatus:=ez202_Status.FT202_Low_Low_Flow_Alarm;		END_IF;
//IF NOT(PVL.s8098[s8098_mapping.FT_202].PDO.VolumeFlow.Status.eStatus=burkert.eSensor_Status.HiHi_Alarm)	THEN	tStatus:=ez202_Status.FT202_High_High_Flow_Alarm;		END_IF;
//IF NOT(PVL.s8098[s8098_mapping.FT_203].PDO.VolumeFlow.Status.eStatus=burkert.eSensor_Status.Low_Low_Alarm)	THEN	tStatus:=ez202_Status.FT203_Low_Low_Flow_Alarm;		END_IF;
//IF NOT(PVL.s8098[s8098_mapping.FT_203].PDO.VolumeFlow.Status.eStatus=burkert.eSensor_Status.HiHi_Alarm)	THEN	tStatus:=ez202_Status.FT202_High_High_Flow_Alarm;		END_IF;

IF (PVL.s8098[s8098_mapping.FT_202].PDO.VolumeFlow.Status.eStatus=burkert.eSensor_Status.Low_Low_Alarm)	THEN	tStatus:=ez202_Status.FT202_Low_Low_Flow_Alarm;		END_IF;
//IF (PVL.s8098[s8098_mapping.FT_202].PDO.VolumeFlow.Status.eStatus=burkert.eSensor_Status.HiHi_Alarm)	THEN	tStatus:=ez202_Status.FT202_High_High_Flow_Alarm;		END_IF;
//IF (PVL.s8098[s8098_mapping.FT_203].PDO.VolumeFlow.Status.eStatus=burkert.eSensor_Status.Low_Low_Alarm)	THEN	tStatus:=ez202_Status.FT203_Low_Low_Flow_Alarm;		END_IF;
//IF (PVL.s8098[s8098_mapping.FT_203].PDO.VolumeFlow.Status.eStatus=burkert.eSensor_Status.HiHi_Alarm)	THEN	tStatus:=ez202_Status.FT202_High_High_Flow_Alarm;		END_IF;


IF PVl.s8312[s8312_mapping.PT_202].Status.eStatus= Burkert.eSensor_Status.HiHi_Alarm THEN tStatus:=eZ202_Status.PT202_High_Pressure_Alarm; END_IF;
IF PVl.s8312[s8312_mapping.PT_202].Status.eStatus= Burkert.eSensor_Status.Low_Low_Alarm THEN tStatus:=eZ202_Status.PT202_Low_Pressure_Alarm; END_IF;
//IF PVl.s8312[s8312_mapping.PT_203].Status.eStatus= Burkert.eSensor_Status.HiHi_Alarm THEN tStatus:=eZ202_Status.PT203_High_Pressure_Alarm; END_IF;
//IF PVl.s8312[s8312_mapping.PT_203].Status.eStatus= Burkert.eSensor_Status.Low_Low_Alarm THEN tStatus:=eZ202_Status.PT203_Low_Pressure_Alarm; END_IF;

Test_Filters_P202:=tStatus;




                
END_METHOD

METHOD Test_Combined : eZ202_Status
  VAR_INPUT
    Status : eZ202_status;
  END_VAR
  VAR
    tStatus : eZ202_Status;
  END_VAR
                  tStatus:=Status;


IF NOT(GVL.s3363[s3363_mapping.ACV_203].Ready) 	THEN 	tStatus:=eZ202_Status.ACV203_Not_Ready; 	END_IF;
IF NOT(GVL.s3363[s3363_mapping.ACV_206].Ready) 	THEN 	tStatus:=eZ202_Status.ACV206_Not_Ready; 	END_IF;
//IF NOT(GVL.s3363[s3363_mapping.ACV_224].Ready) 	THEN 	tStatus:=eZ202_Status.ACV224_Not_Ready; 	END_IF;
//IF NOT(GVL.s3363[s3363_mapping.ACV_225].Ready) 	THEN 	tStatus:=eZ202_Status.ACV225_Not_Ready; 	END_IF;
IF NOT(GVL.s3363[s3363_mapping.ACV_226].Ready) 	THEN 	tStatus:=eZ202_Status.ACV226_Not_Ready; 	END_IF;

IF NOT(Network.VFD[VFD_Mapping.VFD_202].Ready) 	THEN	tStatus:=eZ202_status.P202_Not_Ready;		END_IF;
IF NOT(Network.VFD[VFD_Mapping.VFD_203].Ready) 	THEN	tStatus:=eZ202_status.P203_Not_Ready;		END_IF;

IF NOT(PVL.Ait[AIT_Mapping.LT_202].Ready) 		THEN	tStatus:=eZ202_Status.LT202_Not_Ready;		END_IF;
IF NOT(PVL.Ait[AIT_Mapping.LT_202A].Ready) 		THEN	tStatus:=eZ202_Status.LT202A_Not_Ready;		END_IF;

IF (PVL.Ait[AIT_Mapping.LT_202].Ready) 		THEN	tStatus:=eZ202_Status.LT202_Not_Ready;		END_IF;
IF (PVL.Ait[AIT_Mapping.LT_202].Status.eStatus=Burkert.eSensor_Status.HiHi_Alarm) 		THEN	tStatus:=eZ202_Status.LT202_High_High_Alarm;		END_IF;

IF (PVL.Ait[AIT_Mapping.LT_201].Ready) 		THEN	tStatus:=eZ202_Status.LT201_Not_Ready;		END_IF;
IF (PVL.Ait[AIT_Mapping.LT_201].Status.eStatus=Burkert.eSensor_Status.HiHi_Alarm) 		THEN	tStatus:=eZ202_Status.LT201_High_High_Alarm;		END_IF;

IF (PVL.Ait[AIT_Mapping.LT_101_p].Ready) 		THEN	tStatus:=eZ202_Status.LT101_Not_Ready;		END_IF;
IF (PVL.Ait[AIT_Mapping.LT_101_P].Status.eStatus=Burkert.eSensor_Status.HiHi_Alarm) 		THEN	tStatus:=eZ202_Status.LT101_High_High_Alarm;		END_IF;

IF NOT(PVl.s8312[s8312_mapping.PT_202].Ready)	THEN	tStatus:=ez202_Status.PT202_Not_Ready;		END_IF;
///////********		IF NOT(PVl.s8312[s8312_mapping.PT_203].Ready)	THEN	tStatus:=ez202_Status.PT203_Not_Ready;		END_IF;

IF NOT(PVL.s8098[s8098_mapping.FT_202].Ready)	THEN	tStatus:=ez202_Status.FT202_Not_Ready;		END_IF;
//IF NOT(PVL.s8098[s8098_mapping.FT_203].Ready)	THEN	tStatus:=ez202_Status.FT203_Not_Ready;		END_IF;
	
IF gvl.LS[ls_mapping.LSLL_205].Status.eStatus=Burkert.DI_Status.No_Liquid_Detected_Alarm	THEN	tStatus:=eZ202_Status.P202_Intake_Empty;		END_IF;
IF gvl.LS[ls_mapping.LSLL_203].Status.eStatus=Burkert.DI_Status.No_Liquid_Detected_Alarm	THEN	tStatus:=eZ202_Status.P203_Intake_Empty;		END_IF;
IF gvl.LS[ls_mapping.LSHH_201].Status.eStatus=Burkert.DI_Status.Liquid_Detected_Alarm		THEN	tStatus:=eZ202_Status.EP101_High_High_Alarm;	END_IF;

//IF (PVL.Ait[AIT_Mapping.LT_202].Ready) 		THEN	tStatus:=eZ202_Status.LT202_Not_Ready;		END_IF;
//IF (PVL.Ait[AIT_Mapping.LT_202A].Ready) 		THEN	tStatus:=eZ202_Status.LT202A_Not_Ready;		END_IF;


IF GVL.s3363[s3363_mapping.ACV_203].Status.eStatus=Burkert.eACV_Status.Pos_Error THEN	tStatus:=eZ202_Status.ACV203_Error; END_IF;
IF GVL.s3363[s3363_mapping.ACV_206].Status.eStatus=Burkert.eACV_Status.Pos_Error THEN	tStatus:=eZ202_Status.ACV206_Error; END_IF;
//IF GVL.s3363[s3363_mapping.ACV_224].Status.eStatus=Burkert.eACV_Status.Pos_Error THEN	tStatus:=eZ202_Status.ACV224_Error; END_IF;
//IF GVL.s3363[s3363_mapping.ACV_225].Status.eStatus=Burkert.eACV_Status.Pos_Error THEN	tStatus:=eZ202_Status.ACV225_Error; END_IF;
IF GVL.s3363[s3363_mapping.ACV_226].Status.eStatus=Burkert.eACV_Status.Pos_Error THEN	tStatus:=eZ202_Status.ACV226_Error; END_IF;


//IF NOT(GVL.Filter_Path_Available) THEN tStatus:=eZ202_Status.No_Filter_Available; END_IF;


/////////////////////////////
	

IF NOT(GVL.Filter_Path_Available) THEN tStatus:=eZ202_Status.No_Filter_Available; END_IF;

IF PVL.AIT[AIT_Mapping.LT_202].Status.eStatus=Burkert.eSensor_Status.Low_Low_Alarm THEN	tStatus:=eZ202_Status.LT202_Low_Low_Alarm;	END_IF;
//IF PVL.AIT[AIT_Mapping.LT_202A].Status.eStatus=Burkert.eSensor_Status.Low_Low_Alarm THEN	tStatus:=eZ202_Status.LT202A_Low_Low_Alarm;	END_IF;

IF (PVL.s8098[s8098_mapping.FT_202].PDO.VolumeFlow.Status.eStatus=burkert.eSensor_Status.Low_Low_Alarm)	THEN	tStatus:=ez202_Status.FT202_Low_Low_Flow_Alarm;		END_IF;
//IF (PVL.s8098[s8098_mapping.FT_202].PDO.VolumeFlow.Status.eStatus=burkert.eSensor_Status.HiHi_Alarm)	THEN	tStatus:=ez202_Status.FT202_High_High_Flow_Alarm;		END_IF;
IF (PVL.s8098[s8098_mapping.FT_203].PDO.VolumeFlow.Status.eStatus=burkert.eSensor_Status.Low_Low_Alarm)	THEN	tStatus:=ez202_Status.FT203_Low_Low_Flow_Alarm;		END_IF;
//IF (PVL.s8098[s8098_mapping.FT_203].PDO.VolumeFlow.Status.eStatus=burkert.eSensor_Status.HiHi_Alarm)	THEN	tStatus:=ez202_Status.FT202_High_High_Flow_Alarm;		END_IF;


IF PVl.s8312[s8312_mapping.PT_202].Status.eStatus= Burkert.eSensor_Status.HiHi_Alarm THEN tStatus:=eZ202_Status.PT202_High_Pressure_Alarm; END_IF;
IF PVl.s8312[s8312_mapping.PT_202].Status.eStatus= Burkert.eSensor_Status.Low_Low_Alarm THEN tStatus:=eZ202_Status.PT202_Low_Pressure_Alarm; END_IF;
///////********		IF PVl.s8312[s8312_mapping.PT_203].Status.eStatus= Burkert.eSensor_Status.HiHi_Alarm THEN tStatus:=eZ202_Status.PT203_High_Pressure_Alarm; END_IF;
///////********		IF PVl.s8312[s8312_mapping.PT_203].Status.eStatus= Burkert.eSensor_Status.Low_Low_Alarm THEN tStatus:=eZ202_Status.PT203_Low_Pressure_Alarm; END_IF;

IF NOT(PVL.Ait[AIT_Mapping.LT_202].Ready) 		THEN	tStatus:=eZ202_Status.LT202_Not_Ready;		END_IF;
IF (PVL.Ait[AIT_Mapping.LT_202].Status.eStatus=Burkert.eSensor_Status.HiHi_Alarm) 		THEN	tStatus:=eZ202_Status.LT202_High_High_Alarm;		END_IF;

IF NOT(PVL.Ait[AIT_Mapping.LT_201].Ready) 		THEN	tStatus:=eZ202_Status.LT201_Not_Ready;		END_IF;
IF (PVL.Ait[AIT_Mapping.LT_201].Status.eStatus=Burkert.eSensor_Status.HiHi_Alarm) 		THEN	tStatus:=eZ202_Status.LT201_High_High_Alarm;		END_IF;

IF NOT(PVL.Ait[AIT_Mapping.LT_101_p].Ready) 		THEN	tStatus:=eZ202_Status.LT101_Not_Ready;		END_IF;
IF (PVL.Ait[AIT_Mapping.LT_101_P].Status.eStatus=Burkert.eSensor_Status.HiHi_Alarm) 		THEN	tStatus:=eZ202_Status.LT101_High_High_Alarm;		END_IF;

IF (PVL.Ait[AIT_Mapping.LT_202].Status.eStatus=Burkert.eSensor_Status.Low_Low_Alarm) 		THEN	tStatus:=eZ202_Status.LT202_Low_Low_Alarm;		END_IF;





Test_Combined:=tStatus;
                
END_METHOD

METHOD Test_All : eZ202_Status
  VAR_INPUT
    Status : eZ202_status;
  END_VAR
  VAR
    tStatus : eZ202_Status;
  END_VAR
                  tStatus:=Status;


IF NOT(GVL.s3363[s3363_mapping.ACV_203].Ready) 	THEN 	tStatus:=eZ202_Status.ACV203_Not_Ready; 	END_IF;
IF NOT(GVL.s3363[s3363_mapping.ACV_206].Ready) 	THEN 	tStatus:=eZ202_Status.ACV206_Not_Ready; 	END_IF;
//IF NOT(GVL.s3363[s3363_mapping.ACV_224].Ready) 	THEN 	tStatus:=eZ202_Status.ACV224_Not_Ready; 	END_IF;
//IF NOT(GVL.s3363[s3363_mapping.ACV_225].Ready) 	THEN 	tStatus:=eZ202_Status.ACV225_Not_Ready; 	END_IF;
IF NOT(GVL.s3363[s3363_mapping.ACV_226].Ready) 	THEN 	tStatus:=eZ202_Status.ACV226_Not_Ready; 	END_IF;

IF NOT(Network.VFD[VFD_Mapping.VFD_202].Ready) 	THEN	tStatus:=eZ202_status.P202_Not_Ready;		END_IF;
IF NOT(Network.VFD[VFD_Mapping.VFD_203].Ready) 	THEN	tStatus:=eZ202_status.P203_Not_Ready;		END_IF;

IF NOT(PVL.Ait[AIT_Mapping.LT_202].Ready) 		THEN	tStatus:=eZ202_Status.LT202_Not_Ready;		END_IF;
//IF NOT(PVL.Ait[AIT_Mapping.LT_202A].Ready) 		THEN	tStatus:=eZ202_Status.LT202A_Not_Ready;		END_IF;

IF NOT(PVl.s8312[s8312_mapping.PT_202].Ready)	THEN	tStatus:=ez202_Status.PT202_Not_Ready;		END_IF;
///////********		IF NOT(PVl.s8312[s8312_mapping.PT_203].Ready)	THEN	tStatus:=ez202_Status.PT203_Not_Ready;		END_IF;

IF NOT(PVL.s8098[s8098_mapping.FT_202].Ready)	THEN	tStatus:=ez202_Status.FT202_Not_Ready;		END_IF;
IF NOT(PVL.s8098[s8098_mapping.FT_203].Ready)	THEN	tStatus:=ez202_Status.FT203_Not_Ready;		END_IF;
	
IF gvl.LS[ls_mapping.LSLL_205].Status.eStatus=Burkert.DI_Status.No_Liquid_Detected_Alarm	THEN	tStatus:=eZ202_Status.P202_Intake_Empty;		END_IF;
IF gvl.LS[ls_mapping.LSLL_203].Status.eStatus=Burkert.DI_Status.No_Liquid_Detected_Alarm	THEN	tStatus:=eZ202_Status.P203_Intake_Empty;		END_IF;
IF gvl.LS[ls_mapping.LSHH_201].Status.eStatus=Burkert.DI_Status.Liquid_Detected_Alarm		THEN	tStatus:=eZ202_Status.EP101_High_High_Alarm;	END_IF;

//IF (PVL.Ait[AIT_Mapping.LT_202].Ready) 		THEN	tStatus:=eZ202_Status.LT202_Not_Ready;		END_IF;
//IF (PVL.Ait[AIT_Mapping.LT_202A].Ready) 		THEN	tStatus:=eZ202_Status.LT202A_Not_Ready;		END_IF;


IF GVL.s3363[s3363_mapping.ACV_203].Status.eStatus=Burkert.eACV_Status.Pos_Error THEN	tStatus:=eZ202_Status.ACV203_Error; END_IF;
IF GVL.s3363[s3363_mapping.ACV_206].Status.eStatus=Burkert.eACV_Status.Pos_Error THEN	tStatus:=eZ202_Status.ACV206_Error; END_IF;
//IF GVL.s3363[s3363_mapping.ACV_224].Status.eStatus=Burkert.eACV_Status.Pos_Error THEN	tStatus:=eZ202_Status.ACV224_Error; END_IF;
//IF GVL.s3363[s3363_mapping.ACV_225].Status.eStatus=Burkert.eACV_Status.Pos_Error THEN	tStatus:=eZ202_Status.ACV225_Error; END_IF;
IF GVL.s3363[s3363_mapping.ACV_226].Status.eStatus=Burkert.eACV_Status.Pos_Error THEN	tStatus:=eZ202_Status.ACV226_Error; END_IF;

//IF NOT(GVL.Filter_Path_Available) THEN tStatus:=eZ202_Status.No_Filter_Available; END_IF;

